LIN {X -15.567,Y 120.221,Z 250.000,A 0.000,B 0.000,C 180.000,E1 0.000} C_DIS
LIN {X -9.353,Y 120.863,Z 250.000,A 0.000,B 0.000,C 180.000,E1 0.000} C_DIS
LIN {X -3.119,Y 121.185,Z 250.000,A 0.000,B 0.000,C 180.000,E1 0.000} C_DIS
LIN {X 3.119,Y 121.185,Z 250.000,A 0.000,B 0.000,C 180.000,E1 0.000} C_DIS
LIN {X 4.435,Y 121.117,Z 250.000,A 0.000,B 0.000,C 180.000,E1 0.000} C_DIS
LIN {X 121.110,Y 4.442,Z 250.000,A 0.000,B 0.000,C 180.000,E1 0.000} C_DIS
;rapid-leaky
$VEL.CP=0.3
LIN {X 123.797,Y -61.877,Z 260.000,A 0.000,B 0.000,C 180.000,E1 0.000} C_DIS
;bead-perimeter_outer
$VEL.CP=0.29
LIN {X 126.817,Y -55.423,Z 260.000,A 0.000,B 0.000,C 180.000,E1 0.000} C_DIS
LIN {X 129.503,Y -48.820,Z 260.000,A 0.000,B 0.000,C 180.000,E1 0.000} C_DIS
LIN {X 131.844,Y -42.089,Z 260.000,A 0.000,B 0.000,C 180.000,E1 0.000} C_DIS
LIN {X 133.836,Y -35.246,Z 260.000,A 0.000,B 0.000,C 180.000,E1 0.000} C_DIS
LIN {X 135.473,Y -28.310,Z 260.000,A 0.000,B 0.000,C 180.000,E1 0.000} C_DIS
LIN {X 136.751,Y -21.298,Z 260.000,A 0.000,B 0.000,C 180.000,E1 0.000} C_DIS
LIN {X 137.666,Y -14.230,Z 260.000,A 0.000,B 0.000,C 180.000,E1 0.000} C_DIS
LIN {X 138.216,Y -7.125,Z 260.000,A 0.000,B 0.000,C 180.000,E1 0.000} C_DIS
LIN {X 138.399,Y 0.000,Z 260.000,A 0.000,B 0.000,C 180.000,E1 0.000} C_DIS
LIN {X 138.216,Y 7.125,Z 260.000,A 0.000,B 0.000,C 180.000,E1 0.000} C_DIS
LIN {X 137.666,Y 14.230,Z 260.000,A 0.000,B 0.000,C 180.000,E1 0.000} C_DIS
LIN {X 136.751,Y 21.298,Z 260.000,A 0.000,B 0.000,C 180.000,E1 0.000} C_DIS
LIN {X 135.473,Y 28.310,Z 260.000,A 0.000,B 0.000,C 180.000,E1 0.000} C_DIS
LIN {X 133.836,Y 35.246,Z 260.000,A 0.000,B 0.000,C 180.000,E1 0.000} C_DIS
LIN {X 131.844,Y 42.089,Z 260.000,A 0.000,B 0.000,C 180.000,E1 0.000} C_DIS
LIN {X 129.503,Y 48.820,Z 260.000,A 0.000,B 0.000,C 180.000,E1 0.000} C_DIS
LIN {X 126.817,Y 55.423,Z 260.000,A 0.000,B 0.000,C 180.000,E1 0.000} C_DIS
LIN {X 123.798,Y 61.876,Z 260.000,A 0.000,B 0.000,C 180.000,E1 0.000} C_DIS
LIN {X 120.447,Y 68.168,Z 260.000,A 0.000,B 0.000,C 180.000,E1 0.000} C_DIS
LIN {X 116.778,Y 74.279,Z 260.000,A 0.000,B 0.000,C 180.000,E1 0.000} C_DIS
LIN {X 112.799,Y 80.191,Z 260.000,A 0.000,B 0.000,C 180.000,E1 0.000} C_DIS
LIN {X 108.521,Y 85.892,Z 260.000,A 0.000,B 0.000,C 180.000,E1 0.000} C_DIS
LIN {X 103.956,Y 91.365,Z 260.000,A 0.000,B 0.000,C 180.000,E1 0.000} C_DIS
LIN {X 99.115,Y 96.595,Z 260.000,A 0.000,B 0.000,C 180.000,E1 0.000} C_DIS
LIN {X 94.012,Y 101.569,Z 260.000,A 0.000,B 0.000,C 180.000,E1 0.000} C_DIS
LIN {X 88.657,Y 106.273,Z 260.000,A 0.000,B 0.000,C 180.000,E1 0.000} C_DIS
LIN {X 83.069,Y 110.697,Z 260.000,A 0.000,B 0.000,C 180.000,E1 0.000} C_DIS
LIN {X 77.260,Y 114.827,Z 260.000,A 0.000,B 0.000,C 180.000,E1 0.000} C_DIS
LIN {X 71.246,Y 118.652,Z 260.000,A 0.000,B 0.000,C 180.000,E1 0.000} C_DIS
LIN {X 65.044,Y 122.163,Z 260.000,A 0.000,B 0.000,C 180.000,E1 0.000} C_DIS
LIN {X 58.671,Y 125.348,Z 260.000,A 0.000,B 0.000,C 180.000,E1 0.000} C_DIS
LIN {X 52.139,Y 128.202,Z 260.000,A 0.000,B 0.000,C 180.000,E1 0.000} C_DIS
LIN {X 45.470,Y 130.717,Z 260.000,A 0.000,B 0.000,C 180.000,E1 0.000} C_DIS
LIN {X 38.681,Y 132.884,Z 260.000,A 0.000,B 0.000,C 180.000,E1 0.000} C_DIS
LIN {X 31.788,Y 134.699,Z 260.000,A 0.000,B 0.000,C 180.000,E1 0.000} C_DIS
LIN {X 24.813,Y 136.157,Z 260.000,A 0.000,B 0.000,C 180.000,E1 0.000} C_DIS
LIN {X 17.771,Y 137.253,Z 260.000,A 0.000,B 0.000,C 180.000,E1 0.000} C_DIS
LIN {X 10.681,Y 137.986,Z 260.000,A 0.000,B 0.000,C 180.000,E1 0.000} C_DIS
LIN {X 3.564,Y 138.353,Z 260.000,A 0.000,B 0.000,C 180.000,E1 0.000} C_DIS
LIN {X -3.565,Y 138.353,Z 260.000,A 0.000,B 0.000,C 180.000,E1 0.000} C_DIS
LIN {X -10.680,Y 137.987,Z 260.000,A 0.000,B 0.000,C 180.000,E1 0.000} C_DIS
LIN {X -17.771,Y 137.253,Z 260.000,A 0.000,B 0.000,C 180.000,E1 0.000} C_DIS
LIN {X -24.813,Y 136.157,Z 260.000,A 0.000,B 0.000,C 180.000,E1 0.000} C_DIS
LIN {X -31.788,Y 134.699,Z 260.000,A 0.000,B 0.000,C 180.000,E1 0.000} C_DIS
LIN {X -38.681,Y 132.884,Z 260.000,A 0.000,B 0.000,C 180.000,E1 0.000} C_DIS
LIN {X -45.470,Y 130.717,Z 260.000,A 0.000,B 0.000,C 180.000,E1 0.000} C_DIS
LIN {X -52.139,Y 128.202,Z 260.000,A 0.000,B 0.000,C 180.000,E1 0.000} C_DIS
LIN {X -58.671,Y 125.348,Z 260.000,A 0.000,B 0.000,C 180.000,E1 0.000} C_DIS
LIN {X -65.044,Y 122.163,Z 260.000,A 0.000,B 0.000,C 180.000,E1 0.000} C_DIS
LIN {X -71.246,Y 118.652,Z 260.000,A 0.000,B 0.000,C 180.000,E1 0.000} C_DIS
LIN {X -77.260,Y 114.827,Z 260.000,A 0.000,B 0.000,C 180.000,E1 0.000} C_DIS
LIN {X -83.069,Y 110.697,Z 260.000,A 0.000,B 0.000,C 180.000,E1 0.000} C_DIS
LIN {X -88.657,Y 106.273,Z 260.000,A 0.000,B 0.000,C 180.000,E1 0.000} C_DIS
LIN {X -94.012,Y 101.569,Z 260.000,A 0.000,B 0.000,C 180.000,E1 0.000} C_DIS
LIN {X -99.115,Y 96.595,Z 260.000,A 0.000,B 0.000,C 180.000,E1 0.000} C_DIS
LIN {X -103.956,Y 91.365,Z 260.000,A 0.000,B 0.000,C 180.000,E1 0.000} C_DIS
LIN {X -108.521,Y 85.892,Z 260.000,A 0.000,B 0.000,C 180.000,E1 0.000} C_DIS
LIN {X -112.799,Y 80.191,Z 260.000,A 0.000,B 0.000,C 180.000,E1 0.000} C_DIS
LIN {X -116.778,Y 74.278,Z 260.000,A 0.000,B 0.000,C 180.000,E1 0.000} C_DIS
LIN {X -120.446,Y 68.169,Z 260.000,A 0.000,B 0.000,C 180.000,E1 0.000} C_DIS
LIN {X -123.797,Y 61.877,Z 260.000,A 0.000,B 0.000,C 180.000,E1 0.000} C_DIS
LIN {X -126.817,Y 55.423,Z 260.000,A 0.000,B 0.000,C 180.000,E1 0.000} C_DIS
LIN {X -129.503,Y 48.820,Z 260.000,A 0.000,B 0.000,C 180.000,E1 0.000} C_DIS
LIN {X -131.844,Y 42.089,Z 260.000,A 0.000,B 0.000,C 180.000,E1 0.000} C_DIS
LIN {X -133.836,Y 35.246,Z 260.000,A 0.000,B 0.000,C 180.000,E1 0.000} C_DIS
LIN {X -135.473,Y 28.310,Z 260.000,A 0.000,B 0.000,C 180.000,E1 0.000} C_DIS
LIN {X -136.751,Y 21.298,Z 260.000,A 0.000,B 0.000,C 180.000,E1 0.000} C_DIS
LIN {X -137.666,Y 14.230,Z 260.000,A 0.000,B 0.000,C 180.000,E1 0.000} C_DIS
LIN {X -138.216,Y 7.125,Z 260.000,A 0.000,B 0.000,C 180.000,E1 0.000} C_DIS
LIN {X -138.399,Y 0.000,Z 260.000,A 0.000,B 0.000,C 180.000,E1 0.000} C_DIS
LIN {X -138.216,Y -7.125,Z 260.000,A 0.000,B 0.000,C 180.000,E1 0.000} C_DIS
LIN {X -137.666,Y -14.230,Z 260.000,A 0.000,B 0.000,C 180.000,E1 0.000} C_DIS
LIN {X -136.751,Y -21.298,Z 260.000,A 0.000,B 0.000,C 180.000,E1 0.000} C_DIS
LIN {X -135.473,Y -28.310,Z 260.000,A 0.000,B 0.000,C 180.000,E1 0.000} C_DIS
LIN {X -133.836,Y -35.246,Z 260.000,A 0.000,B 0.000,C 180.000,E1 0.000} C_DIS
LIN {X -131.844,Y -42.089,Z 260.000,A 0.000,B 0.000,C 180.000,E1 0.000} C_DIS
LIN {X -129.503,Y -48.820,Z 260.000,A 0.000,B 0.000,C 180.000,E1 0.000} C_DIS
LIN {X -126.817,Y -55.423,Z 260.000,A 0.000,B 0.000,C 180.000,E1 0.000} C_DIS
LIN {X -123.798,Y -61.876,Z 260.000,A 0.000,B 0.000,C 180.000,E1 0.000} C_DIS
LIN {X -120.447,Y -68.168,Z 260.000,A 0.000,B 0.000,C 180.000,E1 0.000} C_DIS
LIN {X -116.778,Y -74.279,Z 260.000,A 0.000,B 0.000,C 180.000,E1 0.000} C_DIS
LIN {X -112.799,Y -80.191,Z 260.000,A 0.000,B 0.000,C 180.000,E1 0.000} C_DIS
LIN {X -108.521,Y -85.892,Z 260.000,A 0.000,B 0.000,C 180.000,E1 0.000} C_DIS
LIN {X -103.956,Y -91.365,Z 260.000,A 0.000,B 0.000,C 180.000,E1 0.000} C_DIS
LIN {X -99.115,Y -96.595,Z 260.000,A 0.000,B 0.000,C 180.000,E1 0.000} C_DIS
LIN {X -94.012,Y -101.569,Z 260.000,A 0.000,B 0.000,C 180.000,E1 0.000} C_DIS
LIN {X -88.657,Y -106.273,Z 260.000,A 0.000,B 0.000,C 180.000,E1 0.000} C_DIS
LIN {X -83.069,Y -110.697,Z 260.000,A 0.000,B 0.000,C 180.000,E1 0.000} C_DIS
LIN {X -77.260,Y -114.827,Z 260.000,A 0.000,B 0.000,C 180.000,E1 0.000} C_DIS
LIN {X -71.246,Y -118.652,Z 260.000,A 0.000,B 0.000,C 180.000,E1 0.000} C_DIS
LIN {X -65.044,Y -122.163,Z 260.000,A 0.000,B 0.000,C 180.000,E1 0.000} C_DIS
LIN {X -58.671,Y -125.348,Z 260.000,A 0.000,B 0.000,C 180.000,E1 0.000} C_DIS
LIN {X -52.139,Y -128.202,Z 260.000,A 0.000,B 0.000,C 180.000,E1 0.000} C_DIS
LIN {X -45.470,Y -130.717,Z 260.000,A 0.000,B 0.000,C 180.000,E1 0.000} C_DIS
LIN {X -38.681,Y -132.884,Z 260.000,A 0.000,B 0.000,C 180.000,E1 0.000} C_DIS
LIN {X -31.788,Y -134.699,Z 260.000,A 0.000,B 0.000,C 180.000,E1 0.000} C_DIS
LIN {X -24.813,Y -136.157,Z 260.000,A 0.000,B 0.000,C 180.000,E1 0.000} C_DIS
LIN {X -17.771,Y -137.253,Z 260.000,A 0.000,B 0.000,C 180.000,E1 0.000} C_DIS
LIN {X -10.681,Y -137.986,Z 260.000,A 0.000,B 0.000,C 180.000,E1 0.000} C_DIS
LIN {X -3.564,Y -138.353,Z 260.000,A 0.000,B 0.000,C 180.000,E1 0.000} C_DIS
LIN {X 3.565,Y -138.353,Z 260.000,A 0.000,B 0.000,C 180.000,E1 0.000} C_DIS
LIN {X 10.680,Y -137.987,Z 260.000,A 0.000,B 0.000,C 180.000,E1 0.000} C_DIS
LIN {X 17.771,Y -137.253,Z 260.000,A 0.000,B 0.000,C 180.000,E1 0.000} C_DIS
LIN {X 24.813,Y -136.157,Z 260.000,A 0.000,B 0.000,C 180.000,E1 0.000} C_DIS
LIN {X 31.788,Y -134.699,Z 260.000,A 0.000,B 0.000,C 180.000,E1 0.000} C_DIS
LIN {X 38.681,Y -132.884,Z 260.000,A 0.000,B 0.000,C 180.000,E1 0.000} C_DIS
LIN {X 45.470,Y -130.717,Z 260.000,A 0.000,B 0.000,C 180.000,E1 0.000} C_DIS
LIN {X 52.139,Y -128.202,Z 260.000,A 0.000,B 0.000,C 180.000,E1 0.000} C_DIS
LIN {X 58.671,Y -125.348,Z 260.000,A 0.000,B 0.000,C 180.000,E1 0.000} C_DIS
LIN {X 65.044,Y -122.163,Z 260.000,A 0.000,B 0.000,C 180.000,E1 0.000} C_DIS
LIN {X 71.246,Y -118.652,Z 260.000,A 0.000,B 0.000,C 180.000,E1 0.000} C_DIS
LIN {X 77.260,Y -114.827,Z 260.000,A 0.000,B 0.000,C 180.000,E1 0.000} C_DIS
LIN {X 83.069,Y -110.697,Z 260.000,A 0.000,B 0.000,C 180.000,E1 0.000} C_DIS
LIN {X 88.657,Y -106.273,Z 260.000,A 0.000,B 0.000,C 180.000,E1 0.000} C_DIS
LIN {X 94.012,Y -101.569,Z 260.000,A 0.000,B 0.000,C 180.000,E1 0.000} C_DIS
LIN {X 99.115,Y -96.595,Z 260.000,A 0.000,B 0.000,C 180.000,E1 0.000} C_DIS
LIN {X 103.956,Y -91.365,Z 260.000,A 0.000,B 0.000,C 180.000,E1 0.000} C_DIS
LIN {X 108.521,Y -85.892,Z 260.000,A 0.000,B 0.000,C 180.000,E1 0.000} C_DIS
LIN {X 112.799,Y -80.191,Z 260.000,A 0.000,B 0.000,C 180.000,E1 0.000} C_DIS
LIN {X 116.778,Y -74.278,Z 260.000,A 0.000,B 0.000,C 180.000,E1 0.000} C_DIS
LIN {X 120.446,Y -68.169,Z 260.000,A 0.000,B 0.000,C 180.000,E1 0.000} C_DIS
LIN {X 123.797,Y -61.877,Z 260.000,A 0.000,B 0.000,C 180.000,E1 0.000} C_DIS
;rapid-leaky
$VEL.CP=0.3
LIN {X 109.892,Y -54.927,Z 260.000,A 0.000,B 0.000,C 180.000,E1 0.000} C_DIS
;bead-perimeter_inner
$VEL.CP=0.29
LIN {X 112.573,Y -49.198,Z 260.000,A 0.000,B 0.000,C 180.000,E1 0.000} C_DIS
LIN {X 114.957,Y -43.336,Z 260.000,A 0.000,B 0.000,C 180.000,E1 0.000} C_DIS
LIN {X 117.035,Y -37.362,Z 260.000,A 0.000,B 0.000,C 180.000,E1 0.000} C_DIS
LIN {X 118.804,Y -31.287,Z 260.000,A 0.000,B 0.000,C 180.000,E1 0.000} C_DIS
LIN {X 120.256,Y -25.131,Z 260.000,A 0.000,B 0.000,C 180.000,E1 0.000} C_DIS
LIN {X 121.391,Y -18.906,Z 260.000,A 0.000,B 0.000,C 180.000,E1 0.000} C_DIS
LIN {X 122.203,Y -12.631,Z 260.000,A 0.000,B 0.000,C 180.000,E1 0.000} C_DIS
LIN {X 122.691,Y -6.325,Z 260.000,A 0.000,B 0.000,C 180.000,E1 0.000} C_DIS
LIN {X 122.854,Y 0.000,Z 260.000,A 0.000,B 0.000,C 180.000,E1 0.000} C_DIS
LIN {X 122.691,Y 6.325,Z 260.000,A 0.000,B 0.000,C 180.000,E1 0.000} C_DIS
LIN {X 122.203,Y 12.631,Z 260.000,A 0.000,B 0.000,C 180.000,E1 0.000} C_DIS
LIN {X 121.391,Y 18.906,Z 260.000,A 0.000,B 0.000,C 180.000,E1 0.000} C_DIS
LIN {X 120.256,Y 25.131,Z 260.000,A 0.000,B 0.000,C 180.000,E1 0.000} C_DIS
LIN {X 118.804,Y 31.287,Z 260.000,A 0.000,B 0.000,C 180.000,E1 0.000} C_DIS
LIN {X 117.035,Y 37.362,Z 260.000,A 0.000,B 0.000,C 180.000,E1 0.000} C_DIS
LIN {X 114.957,Y 43.336,Z 260.000,A 0.000,B 0.000,C 180.000,E1 0.000} C_DIS
LIN {X 112.572,Y 49.199,Z 260.000,A 0.000,B 0.000,C 180.000,E1 0.000} C_DIS
LIN {X 109.894,Y 54.923,Z 260.000,A 0.000,B 0.000,C 180.000,E1 0.000} C_DIS
LIN {X 106.918,Y 60.511,Z 260.000,A 0.000,B 0.000,C 180.000,E1 0.000} C_DIS
LIN {X 103.661,Y 65.936,Z 260.000,A 0.000,B 0.000,C 180.000,E1 0.000} C_DIS
LIN {X 100.130,Y 71.184,Z 260.000,A 0.000,B 0.000,C 180.000,E1 0.000} C_DIS
LIN {X 96.331,Y 76.246,Z 260.000,A 0.000,B 0.000,C 180.000,E1 0.000} C_DIS
LIN {X 92.280,Y 81.103,Z 260.000,A 0.000,B 0.000,C 180.000,E1 0.000} C_DIS
LIN {X 87.983,Y 85.745,Z 260.000,A 0.000,B 0.000,C 180.000,E1 0.000} C_DIS
LIN {X 83.453,Y 90.160,Z 260.000,A 0.000,B 0.000,C 180.000,E1 0.000} C_DIS
LIN {X 78.700,Y 94.336,Z 260.000,A 0.000,B 0.000,C 180.000,E1 0.000} C_DIS
LIN {X 73.738,Y 98.264,Z 260.000,A 0.000,B 0.000,C 180.000,E1 0.000} C_DIS
LIN {X 68.582,Y 101.929,Z 260.000,A 0.000,B 0.000,C 180.000,E1 0.000} C_DIS
LIN {X 63.243,Y 105.326,Z 260.000,A 0.000,B 0.000,C 180.000,E1 0.000} C_DIS
LIN {X 57.738,Y 108.442,Z 260.000,A 0.000,B 0.000,C 180.000,E1 0.000} C_DIS
LIN {X 52.082,Y 111.268,Z 260.000,A 0.000,B 0.000,C 180.000,E1 0.000} C_DIS
LIN {X 46.283,Y 113.803,Z 260.000,A 0.000,B 0.000,C 180.000,E1 0.000} C_DIS
LIN {X 40.363,Y 116.034,Z 260.000,A 0.000,B 0.000,C 180.000,E1 0.000} C_DIS
LIN {X 34.336,Y 117.958,Z 260.000,A 0.000,B 0.000,C 180.000,E1 0.000} C_DIS
LIN {X 28.217,Y 119.570,Z 260.000,A 0.000,B 0.000,C 180.000,E1 0.000} C_DIS
LIN {X 22.026,Y 120.864,Z 260.000,A 0.000,B 0.000,C 180.000,E1 0.000} C_DIS
LIN {X 15.775,Y 121.837,Z 260.000,A 0.000,B 0.000,C 180.000,E1 0.000} C_DIS
LIN {X 9.481,Y 122.488,Z 260.000,A 0.000,B 0.000,C 180.000,E1 0.000} C_DIS
LIN {X 3.164,Y 122.813,Z 260.000,A 0.000,B 0.000,C 180.000,E1 0.000} C_DIS
LIN {X -3.165,Y 122.813,Z 260.000,A 0.000,B 0.000,C 180.000,E1 0.000} C_DIS
LIN {X -9.479,Y 122.488,Z 260.000,A 0.000,B 0.000,C 180.000,E1 0.000} C_DIS
LIN {X -15.775,Y 121.837,Z 260.000,A 0.000,B 0.000,C 180.000,E1 0.000} C_DIS
LIN {X -22.026,Y 120.864,Z 260.000,A 0.000,B 0.000,C 180.000,E1 0.000} C_DIS
LIN {X -28.217,Y 119.570,Z 260.000,A 0.000,B 0.000,C 180.000,E1 0.000} C_DIS
LIN {X -34.336,Y 117.958,Z 260.000,A 0.000,B 0.000,C 180.000,E1 0.000} C_DIS
LIN {X -40.363,Y 116.034,Z 260.000,A 0.000,B 0.000,C 180.000,E1 0.000} C_DIS
LIN {X -46.283,Y 113.803,Z 260.000,A 0.000,B 0.000,C 180.000,E1 0.000} C_DIS
LIN {X -52.082,Y 111.268,Z 260.000,A 0.000,B 0.000,C 180.000,E1 0.000} C_DIS
LIN {X -57.738,Y 108.442,Z 260.000,A 0.000,B 0.000,C 180.000,E1 0.000} C_DIS
LIN {X -63.243,Y 105.326,Z 260.000,A 0.000,B 0.000,C 180.000,E1 0.000} C_DIS
LIN {X -68.582,Y 101.929,Z 260.000,A 0.000,B 0.000,C 180.000,E1 0.000} C_DIS
LIN {X -73.738,Y 98.264,Z 260.000,A 0.000,B 0.000,C 180.000,E1 0.000} C_DIS
LIN {X -78.700,Y 94.336,Z 260.000,A 0.000,B 0.000,C 180.000,E1 0.000} C_DIS
LIN {X -83.453,Y 90.160,Z 260.000,A 0.000,B 0.000,C 180.000,E1 0.000} C_DIS
LIN {X -87.983,Y 85.745,Z 260.000,A 0.000,B 0.000,C 180.000,E1 0.000} C_DIS
LIN {X -92.280,Y 81.103,Z 260.000,A 0.000,B 0.000,C 180.000,E1 0.000} C_DIS
LIN {X -96.331,Y 76.246,Z 260.000,A 0.000,B 0.000,C 180.000,E1 0.000} C_DIS
LIN {X -100.130,Y 71.184,Z 260.000,A 0.000,B 0.000,C 180.000,E1 0.000} C_DIS
LIN {X -103.662,Y 65.935,Z 260.000,A 0.000,B 0.000,C 180.000,E1 0.000} C_DIS
LIN {X -106.917,Y 60.513,Z 260.000,A 0.000,B 0.000,C 180.000,E1 0.000} C_DIS
LIN {X -109.892,Y 54.927,Z 260.000,A 0.000,B 0.000,C 180.000,E1 0.000} C_DIS
LIN {X -112.573,Y 49.198,Z 260.000,A 0.000,B 0.000,C 180.000,E1 0.000} C_DIS
LIN {X -114.957,Y 43.336,Z 260.000,A 0.000,B 0.000,C 180.000,E1 0.000} C_DIS
LIN {X -117.035,Y 37.362,Z 260.000,A 0.000,B 0.000,C 180.000,E1 0.000} C_DIS
LIN {X -118.804,Y 31.287,Z 260.000,A 0.000,B 0.000,C 180.000,E1 0.000} C_DIS
LIN {X -120.256,Y 25.131,Z 260.000,A 0.000,B 0.000,C 180.000,E1 0.000} C_DIS
LIN {X -121.391,Y 18.906,Z 260.000,A 0.000,B 0.000,C 180.000,E1 0.000} C_DIS
LIN {X -122.203,Y 12.631,Z 260.000,A 0.000,B 0.000,C 180.000,E1 0.000} C_DIS
LIN {X -122.691,Y 6.325,Z 260.000,A 0.000,B 0.000,C 180.000,E1 0.000} C_DIS
LIN {X -122.854,Y 0.000,Z 260.000,A 0.000,B 0.000,C 180.000,E1 0.000} C_DIS
LIN {X -122.691,Y -6.325,Z 260.000,A 0.000,B 0.000,C 180.000,E1 0.000} C_DIS
LIN {X -122.203,Y -12.631,Z 260.000,A 0.000,B 0.000,C 180.000,E1 0.000} C_DIS
LIN {X -121.391,Y -18.906,Z 260.000,A 0.000,B 0.000,C 180.000,E1 0.000} C_DIS
LIN {X -120.256,Y -25.131,Z 260.000,A 0.000,B 0.000,C 180.000,E1 0.000} C_DIS
LIN {X -118.804,Y -31.287,Z 260.000,A 0.000,B 0.000,C 180.000,E1 0.000} C_DIS
LIN {X -117.035,Y -37.362,Z 260.000,A 0.000,B 0.000,C 180.000,E1 0.000} C_DIS
LIN {X -114.957,Y -43.336,Z 260.000,A 0.000,B 0.000,C 180.000,E1 0.000} C_DIS
LIN {X -112.572,Y -49.199,Z 260.000,A 0.000,B 0.000,C 180.000,E1 0.000} C_DIS
LIN {X -109.894,Y -54.923,Z 260.000,A 0.000,B 0.000,C 180.000,E1 0.000} C_DIS
LIN {X -106.918,Y -60.511,Z 260.000,A 0.000,B 0.000,C 180.000,E1 0.000} C_DIS
LIN {X -103.661,Y -65.936,Z 260.000,A 0.000,B 0.000,C 180.000,E1 0.000} C_DIS
LIN {X -100.130,Y -71.184,Z 260.000,A 0.000,B 0.000,C 180.000,E1 0.000} C_DIS
LIN {X -96.331,Y -76.246,Z 260.000,A 0.000,B 0.000,C 180.000,E1 0.000} C_DIS
LIN {X -92.280,Y -81.103,Z 260.000,A 0.000,B 0.000,C 180.000,E1 0.000} C_DIS
LIN {X -87.983,Y -85.745,Z 260.000,A 0.000,B 0.000,C 180.000,E1 0.000} C_DIS
LIN {X -83.453,Y -90.160,Z 260.000,A 0.000,B 0.000,C 180.000,E1 0.000} C_DIS
LIN {X -78.700,Y -94.336,Z 260.000,A 0.000,B 0.000,C 180.000,E1 0.000} C_DIS
LIN {X -73.738,Y -98.264,Z 260.000,A 0.000,B 0.000,C 180.000,E1 0.000} C_DIS
LIN {X -68.582,Y -101.929,Z 260.000,A 0.000,B 0.000,C 180.000,E1 0.000} C_DIS
LIN {X -63.243,Y -105.326,Z 260.000,A 0.000,B 0.000,C 180.000,E1 0.000} C_DIS
LIN {X -57.738,Y -108.442,Z 260.000,A 0.000,B 0.000,C 180.000,E1 0.000} C_DIS
LIN {X -52.082,Y -111.268,Z 260.000,A 0.000,B 0.000,C 180.000,E1 0.000} C_DIS
LIN {X -46.283,Y -113.803,Z 260.000,A 0.000,B 0.000,C 180.000,E1 0.000} C_DIS
LIN {X -40.363,Y -116.034,Z 260.000,A 0.000,B 0.000,C 180.000,E1 0.000} C_DIS
LIN {X -34.336,Y -117.958,Z 260.000,A 0.000,B 0.000,C 180.000,E1 0.000} C_DIS
LIN {X -28.217,Y -119.570,Z 260.000,A 0.000,B 0.000,C 180.000,E1 0.000} C_DIS
LIN {X -22.026,Y -120.864,Z 260.000,A 0.000,B 0.000,C 180.000,E1 0.000} C_DIS
LIN {X -15.775,Y -121.837,Z 260.000,A 0.000,B 0.000,C 180.000,E1 0.000} C_DIS
LIN {X -9.481,Y -122.488,Z 260.000,A 0.000,B 0.000,C 180.000,E1 0.000} C_DIS
LIN {X -3.164,Y -122.813,Z 260.000,A 0.000,B 0.000,C 180.000,E1 0.000} C_DIS
LIN {X 3.165,Y -122.813,Z 260.000,A 0.000,B 0.000,C 180.000,E1 0.000} C_DIS
LIN {X 9.479,Y -122.488,Z 260.000,A 0.000,B 0.000,C 180.000,E1 0.000} C_DIS
LIN {X 15.775,Y -121.837,Z 260.000,A 0.000,B 0.000,C 180.000,E1 0.000} C_DIS
LIN {X 22.026,Y -120.864,Z 260.000,A 0.000,B 0.000,C 180.000,E1 0.000} C_DIS
LIN {X 28.217,Y -119.570,Z 260.000,A 0.000,B 0.000,C 180.000,E1 0.000} C_DIS
LIN {X 34.336,Y -117.958,Z 260.000,A 0.000,B 0.000,C 180.000,E1 0.000} C_DIS
LIN {X 40.363,Y -116.034,Z 260.000,A 0.000,B 0.000,C 180.000,E1 0.000} C_DIS
LIN {X 46.283,Y -113.803,Z 260.000,A 0.000,B 0.000,C 180.000,E1 0.000} C_DIS
LIN {X 52.082,Y -111.268,Z 260.000,A 0.000,B 0.000,C 180.000,E1 0.000} C_DIS
LIN {X 57.738,Y -108.442,Z 260.000,A 0.000,B 0.000,C 180.000,E1 0.000} C_DIS
LIN {X 63.243,Y -105.326,Z 260.000,A 0.000,B 0.000,C 180.000,E1 0.000} C_DIS
LIN {X 68.582,Y -101.929,Z 260.000,A 0.000,B 0.000,C 180.000,E1 0.000} C_DIS
LIN {X 73.738,Y -98.264,Z 260.000,A 0.000,B 0.000,C 180.000,E1 0.000} C_DIS
LIN {X 78.700,Y -94.336,Z 260.000,A 0.000,B 0.000,C 180.000,E1 0.000} C_DIS
LIN {X 83.453,Y -90.160,Z 260.000,A 0.000,B 0.000,C 180.000,E1 0.000} C_DIS
LIN {X 87.983,Y -85.745,Z 260.000,A 0.000,B 0.000,C 180.000,E1 0.000} C_DIS
LIN {X 92.280,Y -81.103,Z 260.000,A 0.000,B 0.000,C 180.000,E1 0.000} C_DIS
LIN {X 96.331,Y -76.246,Z 260.000,A 0.000,B 0.000,C 180.000,E1 0.000} C_DIS
LIN {X 100.130,Y -71.184,Z 260.000,A 0.000,B 0.000,C 180.000,E1 0.000} C_DIS
LIN {X 103.662,Y -65.935,Z 260.000,A 0.000,B 0.000,C 180.000,E1 0.000} C_DIS
LIN {X 106.917,Y -60.513,Z 260.000,A 0.000,B 0.000,C 180.000,E1 0.000} C_DIS
LIN {X 109.892,Y -54.927,Z 260.000,A 0.000,B 0.000,C 180.000,E1 0.000} C_DIS
;rapid-leaky
$VEL.CP=0.3
LIN {X 102.499,Y -23.053,Z 260.000,A 0.000,B 0.000,C 180.000,E1 0.000} C_DIS
;bead-sparse_infill
$VEL.CP=0.29
LIN {X 23.045,Y -102.507,Z 260.000,A 0.000,B 0.000,C 180.000,E1 0.000} C_DIS
LIN {X 18.842,Y -103.386,Z 260.000,A 0.000,B 0.000,C 180.000,E1 0.000} C_DIS
LIN {X 13.494,Y -104.218,Z 260.000,A 0.000,B 0.000,C 180.000,E1 0.000} C_DIS
LIN {X 8.108,Y -104.775,Z 260.000,A 0.000,B 0.000,C 180.000,E1 0.000} C_DIS
LIN {X 2.708,Y -105.053,Z 260.000,A 0.000,B 0.000,C 180.000,E1 0.000} C_DIS
LIN {X -2.707,Y -105.053,Z 260.000,A 0.000,B 0.000,C 180.000,E1 0.000} C_DIS
LIN {X -8.110,Y -104.775,Z 260.000,A 0.000,B 0.000,C 180.000,E1 0.000} C_DIS
LIN {X -13.494,Y -104.218,Z 260.000,A 0.000,B 0.000,C 180.000,E1 0.000} C_DIS
LIN {X -18.842,Y -103.386,Z 260.000,A 0.000,B 0.000,C 180.000,E1 0.000} C_DIS
LIN {X -24.136,Y -102.279,Z 260.000,A 0.000,B 0.000,C 180.000,E1 0.000} C_DIS
LIN {X -29.371,Y -100.900,Z 260.000,A 0.000,B 0.000,C 180.000,E1 0.000} C_DIS
LIN {X -34.526,Y -99.255,Z 260.000,A 0.000,B 0.000,C 180.000,E1 0.000} C_DIS
LIN {X -39.590,Y -97.346,Z 260.000,A 0.000,B 0.000,C 180.000,E1 0.000} C_DIS
LIN {X -44.551,Y -95.177,Z 260.000,A 0.000,B 0.000,C 180.000,E1 0.000} C_DIS
LIN {X -49.389,Y -92.760,Z 260.000,A 0.000,B 0.000,C 180.000,E1 0.000} C_DIS
LIN {X -54.096,Y -90.095,Z 260.000,A 0.000,B 0.000,C 180.000,E1 0.000} C_DIS
LIN {X -58.665,Y -87.189,Z 260.000,A 0.000,B 0.000,C 180.000,E1 0.000} C_DIS
LIN {X -63.074,Y -84.054,Z 260.000,A 0.000,B 0.000,C 180.000,E1 0.000} C_DIS
LIN {X -67.320,Y -80.694,Z 260.000,A 0.000,B 0.000,C 180.000,E1 0.000} C_DIS
LIN {X -71.386,Y -77.121,Z 260.000,A 0.000,B 0.000,C 180.000,E1 0.000} C_DIS
LIN {X -75.260,Y -73.346,Z 260.000,A 0.000,B 0.000,C 180.000,E1 0.000} C_DIS
LIN {X -78.935,Y -69.375,Z 260.000,A 0.000,B 0.000,C 180.000,E1 0.000} C_DIS
LIN {X -82.400,Y -65.221,Z 260.000,A 0.000,B 0.000,C 180.000,E1 0.000} C_DIS
LIN {X -85.650,Y -60.889,Z 260.000,A 0.000,B 0.000,C 180.000,E1 0.000} C_DIS
LIN {X -88.331,Y -56.905,Z 260.000,A 0.000,B 0.000,C 180.000,E1 0.000} C_DIS
LIN {X 56.891,Y 88.317,Z 260.000,A 0.000,B 0.000,C 180.000,E1 0.000} C_DIS
;rapid-leaky
$VEL.CP=0.3
LIN {X 93.706,Y -74.165,Z 270.000,A 0.000,B 0.000,C 180.000,E1 0.000} C_DIS
;bead-perimeter_outer
$VEL.CP=0.21
LIN {X 97.399,Y -69.244,Z 270.000,A 0.000,B 0.000,C 180.000,E1 0.000} C_DIS
LIN {X 100.834,Y -64.137,Z 270.000,A 0.000,B 0.000,C 180.000,E1 0.000} C_DIS
LIN {X 104.003,Y -58.861,Z 270.000,A 0.000,B 0.000,C 180.000,E1 0.000} C_DIS
LIN {X 106.895,Y -53.430,Z 270.000,A 0.000,B 0.000,C 180.000,E1 0.000} C_DIS
LIN {X 109.504,Y -47.856,Z 270.000,A 0.000,B 0.000,C 180.000,E1 0.000} C_DIS
LIN {X 111.822,Y -42.155,Z 270.000,A 0.000,B 0.000,C 180.000,E1 0.000} C_DIS
LIN {X 113.844,Y -36.344,Z 270.000,A 0.000,B 0.000,C 180.000,E1 0.000} C_DIS
LIN {X 115.563,Y -30.435,Z 270.000,A 0.000,B 0.000,C 180.000,E1 0.000} C_DIS
LIN {X 116.977,Y -24.445,Z 270.000,A 0.000,B 0.000,C 180.000,E1 0.000} C_DIS
LIN {X 118.080,Y -18.390,Z 270.000,A 0.000,B 0.000,C 180.000,E1 0.000} C_DIS
LIN {X 118.870,Y -12.288,Z 270.000,A 0.000,B 0.000,C 180.000,E1 0.000} C_DIS
LIN {X 119.346,Y -6.144,Z 270.000,A 0.000,B 0.000,C 180.000,E1 0.000} C_DIS
LIN {X 119.356,Y -5.765,Z 270.000,A 0.000,B 0.000,C 180.000,E1 0.000} C_DIS
LIN {X 119.503,Y -0.001,Z 270.000,A 0.000,B 0.000,C 180.000,E1 0.000} C_DIS
LIN {X 119.345,Y 6.152,Z 270.000,A 0.000,B 0.000,C 180.000,E1 0.000} C_DIS
LIN {X 118.870,Y 12.288,Z 270.000,A 0.000,B 0.000,C 180.000,E1 0.000} C_DIS
LIN {X 118.080,Y 18.390,Z 270.000,A 0.000,B 0.000,C 180.000,E1 0.000} C_DIS
LIN {X 116.977,Y 24.445,Z 270.000,A 0.000,B 0.000,C 180.000,E1 0.000} C_DIS
LIN {X 115.563,Y 30.435,Z 270.000,A 0.000,B 0.000,C 180.000,E1 0.000} C_DIS
LIN {X 113.844,Y 36.344,Z 270.000,A 0.000,B 0.000,C 180.000,E1 0.000} C_DIS
LIN {X 111.822,Y 42.155,Z 270.000,A 0.000,B 0.000,C 180.000,E1 0.000} C_DIS
LIN {X 109.504,Y 47.856,Z 270.000,A 0.000,B 0.000,C 180.000,E1 0.000} C_DIS
LIN {X 106.895,Y 53.430,Z 270.000,A 0.000,B 0.000,C 180.000,E1 0.000} C_DIS
LIN {X 104.003,Y 58.861,Z 270.000,A 0.000,B 0.000,C 180.000,E1 0.000} C_DIS
LIN {X 100.834,Y 64.137,Z 270.000,A 0.000,B 0.000,C 180.000,E1 0.000} C_DIS
LIN {X 97.399,Y 69.244,Z 270.000,A 0.000,B 0.000,C 180.000,E1 0.000} C_DIS
LIN {X 93.706,Y 74.165,Z 270.000,A 0.000,B 0.000,C 180.000,E1 0.000} C_DIS
LIN {X 89.762,Y 78.891,Z 270.000,A 0.000,B 0.000,C 180.000,E1 0.000} C_DIS
LIN {X 85.583,Y 83.407,Z 270.000,A 0.000,B 0.000,C 180.000,E1 0.000} C_DIS
LIN {X 81.176,Y 87.702,Z 270.000,A 0.000,B 0.000,C 180.000,E1 0.000} C_DIS
LIN {X 76.553,Y 91.765,Z 270.000,A 0.000,B 0.000,C 180.000,E1 0.000} C_DIS
LIN {X 71.727,Y 95.584,Z 270.000,A 0.000,B 0.000,C 180.000,E1 0.000} C_DIS
LIN {X 66.712,Y 99.150,Z 270.000,A 0.000,B 0.000,C 180.000,E1 0.000} C_DIS
LIN {X 61.520,Y 102.453,Z 270.000,A 0.000,B 0.000,C 180.000,E1 0.000} C_DIS
LIN {X 56.163,Y 105.484,Z 270.000,A 0.000,B 0.000,C 180.000,E1 0.000} C_DIS
LIN {X 50.660,Y 108.235,Z 270.000,A 0.000,B 0.000,C 180.000,E1 0.000} C_DIS
LIN {X 45.022,Y 110.699,Z 270.000,A 0.000,B 0.000,C 180.000,E1 0.000} C_DIS
LIN {X 39.262,Y 112.870,Z 270.000,A 0.000,B 0.000,C 180.000,E1 0.000} C_DIS
LIN {X 33.399,Y 114.742,Z 270.000,A 0.000,B 0.000,C 180.000,E1 0.000} C_DIS
LIN {X 27.448,Y 116.309,Z 270.000,A 0.000,B 0.000,C 180.000,E1 0.000} C_DIS
LIN {X 21.424,Y 117.568,Z 270.000,A 0.000,B 0.000,C 180.000,E1 0.000} C_DIS
LIN {X 15.345,Y 118.515,Z 270.000,A 0.000,B 0.000,C 180.000,E1 0.000} C_DIS
LIN {X 9.223,Y 119.147,Z 270.000,A 0.000,B 0.000,C 180.000,E1 0.000} C_DIS
LIN {X 3.077,Y 119.464,Z 270.000,A 0.000,B 0.000,C 180.000,E1 0.000} C_DIS
LIN {X -3.079,Y 119.464,Z 270.000,A 0.000,B 0.000,C 180.000,E1 0.000} C_DIS
LIN {X -3.458,Y 119.445,Z 270.000,A 0.000,B 0.000,C 180.000,E1 0.000} C_DIS
LIN {X -9.223,Y 119.147,Z 270.000,A 0.000,B 0.000,C 180.000,E1 0.000} C_DIS
LIN {X -15.345,Y 118.515,Z 270.000,A 0.000,B 0.000,C 180.000,E1 0.000} C_DIS
LIN {X -21.424,Y 117.568,Z 270.000,A 0.000,B 0.000,C 180.000,E1 0.000} C_DIS
LIN {X -27.448,Y 116.309,Z 270.000,A 0.000,B 0.000,C 180.000,E1 0.000} C_DIS
LIN {X -33.399,Y 114.742,Z 270.000,A 0.000,B 0.000,C 180.000,E1 0.000} C_DIS
LIN {X -39.262,Y 112.870,Z 270.000,A 0.000,B 0.000,C 180.000,E1 0.000} C_DIS
LIN {X -45.022,Y 110.699,Z 270.000,A 0.000,B 0.000,C 180.000,E1 0.000} C_DIS
LIN {X -50.660,Y 108.235,Z 270.000,A 0.000,B 0.000,C 180.000,E1 0.000} C_DIS
LIN {X -56.163,Y 105.484,Z 270.000,A 0.000,B 0.000,C 180.000,E1 0.000} C_DIS
LIN {X -61.520,Y 102.453,Z 270.000,A 0.000,B 0.000,C 180.000,E1 0.000} C_DIS
LIN {X -66.712,Y 99.150,Z 270.000,A 0.000,B 0.000,C 180.000,E1 0.000} C_DIS
LIN {X -71.727,Y 95.584,Z 270.000,A 0.000,B 0.000,C 180.000,E1 0.000} C_DIS
LIN {X -76.553,Y 91.765,Z 270.000,A 0.000,B 0.000,C 180.000,E1 0.000} C_DIS
LIN {X -81.176,Y 87.702,Z 270.000,A 0.000,B 0.000,C 180.000,E1 0.000} C_DIS
LIN {X -85.583,Y 83.407,Z 270.000,A 0.000,B 0.000,C 180.000,E1 0.000} C_DIS
LIN {X -89.762,Y 78.891,Z 270.000,A 0.000,B 0.000,C 180.000,E1 0.000} C_DIS
LIN {X -93.706,Y 74.165,Z 270.000,A 0.000,B 0.000,C 180.000,E1 0.000} C_DIS
LIN {X -97.399,Y 69.244,Z 270.000,A 0.000,B 0.000,C 180.000,E1 0.000} C_DIS
LIN {X -100.834,Y 64.137,Z 270.000,A 0.000,B 0.000,C 180.000,E1 0.000} C_DIS
LIN {X -104.003,Y 58.861,Z 270.000,A 0.000,B 0.000,C 180.000,E1 0.000} C_DIS
LIN {X -106.895,Y 53.430,Z 270.000,A 0.000,B 0.000,C 180.000,E1 0.000} C_DIS
LIN {X -109.504,Y 47.856,Z 270.000,A 0.000,B 0.000,C 180.000,E1 0.000} C_DIS
LIN {X -111.822,Y 42.155,Z 270.000,A 0.000,B 0.000,C 180.000,E1 0.000} C_DIS
LIN {X -113.844,Y 36.344,Z 270.000,A 0.000,B 0.000,C 180.000,E1 0.000} C_DIS
LIN {X -115.563,Y 30.435,Z 270.000,A 0.000,B 0.000,C 180.000,E1 0.000} C_DIS
LIN {X -116.977,Y 24.445,Z 270.000,A 0.000,B 0.000,C 180.000,E1 0.000} C_DIS
LIN {X -118.080,Y 18.390,Z 270.000,A 0.000,B 0.000,C 180.000,E1 0.000} C_DIS
LIN {X -118.870,Y 12.288,Z 270.000,A 0.000,B 0.000,C 180.000,E1 0.000} C_DIS
LIN {X -119.346,Y 6.144,Z 270.000,A 0.000,B 0.000,C 180.000,E1 0.000} C_DIS
LIN {X -119.356,Y 5.765,Z 270.000,A 0.000,B 0.000,C 180.000,E1 0.000} C_DIS
LIN {X -119.503,Y 0.001,Z 270.000,A 0.000,B 0.000,C 180.000,E1 0.000} C_DIS
LIN {X -119.345,Y -6.152,Z 270.000,A 0.000,B 0.000,C 180.000,E1 0.000} C_DIS
LIN {X -118.870,Y -12.288,Z 270.000,A 0.000,B 0.000,C 180.000,E1 0.000} C_DIS
LIN {X -118.080,Y -18.390,Z 270.000,A 0.000,B 0.000,C 180.000,E1 0.000} C_DIS
LIN {X -116.977,Y -24.445,Z 270.000,A 0.000,B 0.000,C 180.000,E1 0.000} C_DIS
LIN {X -115.563,Y -30.435,Z 270.000,A 0.000,B 0.000,C 180.000,E1 0.000} C_DIS
LIN {X -113.844,Y -36.344,Z 270.000,A 0.000,B 0.000,C 180.000,E1 0.000} C_DIS
LIN {X -111.822,Y -42.155,Z 270.000,A 0.000,B 0.000,C 180.000,E1 0.000} C_DIS
LIN {X -109.504,Y -47.856,Z 270.000,A 0.000,B 0.000,C 180.000,E1 0.000} C_DIS
LIN {X -106.895,Y -53.430,Z 270.000,A 0.000,B 0.000,C 180.000,E1 0.000} C_DIS
LIN {X -104.003,Y -58.861,Z 270.000,A 0.000,B 0.000,C 180.000,E1 0.000} C_DIS
LIN {X -100.834,Y -64.137,Z 270.000,A 0.000,B 0.000,C 180.000,E1 0.000} C_DIS
LIN {X -97.399,Y -69.244,Z 270.000,A 0.000,B 0.000,C 180.000,E1 0.000} C_DIS
LIN {X -93.706,Y -74.165,Z 270.000,A 0.000,B 0.000,C 180.000,E1 0.000} C_DIS
LIN {X -89.762,Y -78.891,Z 270.000,A 0.000,B 0.000,C 180.000,E1 0.000} C_DIS
LIN {X -85.583,Y -83.407,Z 270.000,A 0.000,B 0.000,C 180.000,E1 0.000} C_DIS
LIN {X -81.176,Y -87.702,Z 270.000,A 0.000,B 0.000,C 180.000,E1 0.000} C_DIS
LIN {X -76.553,Y -91.765,Z 270.000,A 0.000,B 0.000,C 180.000,E1 0.000} C_DIS
LIN {X -71.727,Y -95.584,Z 270.000,A 0.000,B 0.000,C 180.000,E1 0.000} C_DIS
LIN {X -66.712,Y -99.150,Z 270.000,A 0.000,B 0.000,C 180.000,E1 0.000} C_DIS
LIN {X -61.520,Y -102.453,Z 270.000,A 0.000,B 0.000,C 180.000,E1 0.000} C_DIS
LIN {X -56.163,Y -105.484,Z 270.000,A 0.000,B 0.000,C 180.000,E1 0.000} C_DIS
LIN {X -50.660,Y -108.235,Z 270.000,A 0.000,B 0.000,C 180.000,E1 0.000} C_DIS
LIN {X -45.022,Y -110.699,Z 270.000,A 0.000,B 0.000,C 180.000,E1 0.000} C_DIS
LIN {X -39.262,Y -112.870,Z 270.000,A 0.000,B 0.000,C 180.000,E1 0.000} C_DIS
LIN {X -33.399,Y -114.742,Z 270.000,A 0.000,B 0.000,C 180.000,E1 0.000} C_DIS
LIN {X -27.448,Y -116.309,Z 270.000,A 0.000,B 0.000,C 180.000,E1 0.000} C_DIS
LIN {X -21.424,Y -117.568,Z 270.000,A 0.000,B 0.000,C 180.000,E1 0.000} C_DIS
LIN {X -15.345,Y -118.515,Z 270.000,A 0.000,B 0.000,C 180.000,E1 0.000} C_DIS
LIN {X -9.223,Y -119.147,Z 270.000,A 0.000,B 0.000,C 180.000,E1 0.000} C_DIS
LIN {X -3.077,Y -119.464,Z 270.000,A 0.000,B 0.000,C 180.000,E1 0.000} C_DIS
LIN {X 3.079,Y -119.464,Z 270.000,A 0.000,B 0.000,C 180.000,E1 0.000} C_DIS
LIN {X 9.223,Y -119.147,Z 270.000,A 0.000,B 0.000,C 180.000,E1 0.000} C_DIS
LIN {X 15.345,Y -118.515,Z 270.000,A 0.000,B 0.000,C 180.000,E1 0.000} C_DIS
LIN {X 21.424,Y -117.568,Z 270.000,A 0.000,B 0.000,C 180.000,E1 0.000} C_DIS
LIN {X 27.448,Y -116.309,Z 270.000,A 0.000,B 0.000,C 180.000,E1 0.000} C_DIS
LIN {X 33.399,Y -114.742,Z 270.000,A 0.000,B 0.000,C 180.000,E1 0.000} C_DIS
LIN {X 39.262,Y -112.870,Z 270.000,A 0.000,B 0.000,C 180.000,E1 0.000} C_DIS
LIN {X 45.022,Y -110.699,Z 270.000,A 0.000,B 0.000,C 180.000,E1 0.000} C_DIS
LIN {X 50.660,Y -108.235,Z 270.000,A 0.000,B 0.000,C 180.000,E1 0.000} C_DIS
LIN {X 56.163,Y -105.484,Z 270.000,A 0.000,B 0.000,C 180.000,E1 0.000} C_DIS
LIN {X 61.520,Y -102.453,Z 270.000,A 0.000,B 0.000,C 180.000,E1 0.000} C_DIS
LIN {X 66.712,Y -99.150,Z 270.000,A 0.000,B 0.000,C 180.000,E1 0.000} C_DIS
LIN {X 71.727,Y -95.584,Z 270.000,A 0.000,B 0.000,C 180.000,E1 0.000} C_DIS
LIN {X 76.553,Y -91.765,Z 270.000,A 0.000,B 0.000,C 180.000,E1 0.000} C_DIS
LIN {X 81.176,Y -87.702,Z 270.000,A 0.000,B 0.000,C 180.000,E1 0.000} C_DIS
LIN {X 85.583,Y -83.407,Z 270.000,A 0.000,B 0.000,C 180.000,E1 0.000} C_DIS
LIN {X 89.762,Y -78.891,Z 270.000,A 0.000,B 0.000,C 180.000,E1 0.000} C_DIS
LIN {X 93.706,Y -74.165,Z 270.000,A 0.000,B 0.000,C 180.000,E1 0.000} C_DIS
;rapid-leaky
$VEL.CP=0.3
LIN {X 81.517,Y -64.517,Z 270.000,A 0.000,B 0.000,C 180.000,E1 0.000} C_DIS
;bead-perimeter_inner
$VEL.CP=0.21
LIN {X 84.729,Y -60.237,Z 270.000,A 0.000,B 0.000,C 180.000,E1 0.000} C_DIS
LIN {X 87.718,Y -55.794,Z 270.000,A 0.000,B 0.000,C 180.000,E1 0.000} C_DIS
LIN {X 90.475,Y -51.203,Z 270.000,A 0.000,B 0.000,C 180.000,E1 0.000} C_DIS
LIN {X 92.990,Y -46.480,Z 270.000,A 0.000,B 0.000,C 180.000,E1 0.000} C_DIS
LIN {X 95.259,Y -41.630,Z 270.000,A 0.000,B 0.000,C 180.000,E1 0.000} C_DIS
LIN {X 97.277,Y -36.670,Z 270.000,A 0.000,B 0.000,C 180.000,E1 0.000} C_DIS
LIN {X 99.035,Y -31.616,Z 270.000,A 0.000,B 0.000,C 180.000,E1 0.000} C_DIS
LIN {X 100.531,Y -26.477,Z 270.000,A 0.000,B 0.000,C 180.000,E1 0.000} C_DIS
LIN {X 101.760,Y -21.266,Z 270.000,A 0.000,B 0.000,C 180.000,E1 0.000} C_DIS
LIN {X 102.720,Y -15.999,Z 270.000,A 0.000,B 0.000,C 180.000,E1 0.000} C_DIS
LIN {X 103.407,Y -10.689,Z 270.000,A 0.000,B 0.000,C 180.000,E1 0.000} C_DIS
LIN {X 103.822,Y -5.335,Z 270.000,A 0.000,B 0.000,C 180.000,E1 0.000} C_DIS
LIN {X 103.958,Y -0.002,Z 270.000,A 0.000,B 0.000,C 180.000,E1 0.000} C_DIS
LIN {X 103.820,Y 5.352,Z 270.000,A 0.000,B 0.000,C 180.000,E1 0.000} C_DIS
LIN {X 103.407,Y 10.689,Z 270.000,A 0.000,B 0.000,C 180.000,E1 0.000} C_DIS
LIN {X 102.720,Y 15.999,Z 270.000,A 0.000,B 0.000,C 180.000,E1 0.000} C_DIS
LIN {X 101.760,Y 21.266,Z 270.000,A 0.000,B 0.000,C 180.000,E1 0.000} C_DIS
LIN {X 100.531,Y 26.477,Z 270.000,A 0.000,B 0.000,C 180.000,E1 0.000} C_DIS
LIN {X 99.035,Y 31.616,Z 270.000,A 0.000,B 0.000,C 180.000,E1 0.000} C_DIS
LIN {X 97.277,Y 36.670,Z 270.000,A 0.000,B 0.000,C 180.000,E1 0.000} C_DIS
LIN {X 95.259,Y 41.630,Z 270.000,A 0.000,B 0.000,C 180.000,E1 0.000} C_DIS
LIN {X 92.990,Y 46.480,Z 270.000,A 0.000,B 0.000,C 180.000,E1 0.000} C_DIS
LIN {X 90.475,Y 51.203,Z 270.000,A 0.000,B 0.000,C 180.000,E1 0.000} C_DIS
LIN {X 87.718,Y 55.794,Z 270.000,A 0.000,B 0.000,C 180.000,E1 0.000} C_DIS
LIN {X 84.729,Y 60.237,Z 270.000,A 0.000,B 0.000,C 180.000,E1 0.000} C_DIS
LIN {X 81.517,Y 64.517,Z 270.000,A 0.000,B 0.000,C 180.000,E1 0.000} C_DIS
LIN {X 78.086,Y 68.629,Z 270.000,A 0.000,B 0.000,C 180.000,E1 0.000} C_DIS
LIN {X 74.450,Y 72.558,Z 270.000,A 0.000,B 0.000,C 180.000,E1 0.000} C_DIS
LIN {X 70.617,Y 76.293,Z 270.000,A 0.000,B 0.000,C 180.000,E1 0.000} C_DIS
LIN {X 66.595,Y 79.828,Z 270.000,A 0.000,B 0.000,C 180.000,E1 0.000} C_DIS
LIN {X 62.397,Y 83.150,Z 270.000,A 0.000,B 0.000,C 180.000,E1 0.000} C_DIS
LIN {X 58.033,Y 86.253,Z 270.000,A 0.000,B 0.000,C 180.000,E1 0.000} C_DIS
LIN {X 53.517,Y 89.126,Z 270.000,A 0.000,B 0.000,C 180.000,E1 0.000} C_DIS
LIN {X 48.857,Y 91.763,Z 270.000,A 0.000,B 0.000,C 180.000,E1 0.000} C_DIS
LIN {X 44.070,Y 94.156,Z 270.000,A 0.000,B 0.000,C 180.000,E1 0.000} C_DIS
LIN {X 39.167,Y 96.299,Z 270.000,A 0.000,B 0.000,C 180.000,E1 0.000} C_DIS
LIN {X 34.155,Y 98.187,Z 270.000,A 0.000,B 0.000,C 180.000,E1 0.000} C_DIS
LIN {X 29.054,Y 99.817,Z 270.000,A 0.000,B 0.000,C 180.000,E1 0.000} C_DIS
LIN {X 23.878,Y 101.180,Z 270.000,A 0.000,B 0.000,C 180.000,E1 0.000} C_DIS
LIN {X 18.637,Y 102.275,Z 270.000,A 0.000,B 0.000,C 180.000,E1 0.000} C_DIS
LIN {X 13.349,Y 103.099,Z 270.000,A 0.000,B 0.000,C 180.000,E1 0.000} C_DIS
LIN {X 8.024,Y 103.649,Z 270.000,A 0.000,B 0.000,C 180.000,E1 0.000} C_DIS
LIN {X 2.677,Y 103.924,Z 270.000,A 0.000,B 0.000,C 180.000,E1 0.000} C_DIS
LIN {X -2.682,Y 103.924,Z 270.000,A 0.000,B 0.000,C 180.000,E1 0.000} C_DIS
LIN {X -8.023,Y 103.649,Z 270.000,A 0.000,B 0.000,C 180.000,E1 0.000} C_DIS
LIN {X -13.349,Y 103.099,Z 270.000,A 0.000,B 0.000,C 180.000,E1 0.000} C_DIS
LIN {X -18.637,Y 102.275,Z 270.000,A 0.000,B 0.000,C 180.000,E1 0.000} C_DIS
LIN {X -23.878,Y 101.180,Z 270.000,A 0.000,B 0.000,C 180.000,E1 0.000} C_DIS
LIN {X -29.054,Y 99.817,Z 270.000,A 0.000,B 0.000,C 180.000,E1 0.000} C_DIS
LIN {X -34.155,Y 98.187,Z 270.000,A 0.000,B 0.000,C 180.000,E1 0.000} C_DIS
LIN {X -39.167,Y 96.299,Z 270.000,A 0.000,B 0.000,C 180.000,E1 0.000} C_DIS
LIN {X -44.070,Y 94.156,Z 270.000,A 0.000,B 0.000,C 180.000,E1 0.000} C_DIS
LIN {X -48.857,Y 91.763,Z 270.000,A 0.000,B 0.000,C 180.000,E1 0.000} C_DIS
LIN {X -53.517,Y 89.126,Z 270.000,A 0.000,B 0.000,C 180.000,E1 0.000} C_DIS
LIN {X -58.033,Y 86.253,Z 270.000,A 0.000,B 0.000,C 180.000,E1 0.000} C_DIS
LIN {X -62.397,Y 83.150,Z 270.000,A 0.000,B 0.000,C 180.000,E1 0.000} C_DIS
LIN {X -66.595,Y 79.828,Z 270.000,A 0.000,B 0.000,C 180.000,E1 0.000} C_DIS
LIN {X -70.617,Y 76.293,Z 270.000,A 0.000,B 0.000,C 180.000,E1 0.000} C_DIS
LIN {X -74.450,Y 72.558,Z 270.000,A 0.000,B 0.000,C 180.000,E1 0.000} C_DIS
LIN {X -78.086,Y 68.629,Z 270.000,A 0.000,B 0.000,C 180.000,E1 0.000} C_DIS
LIN {X -81.517,Y 64.517,Z 270.000,A 0.000,B 0.000,C 180.000,E1 0.000} C_DIS
LIN {X -84.729,Y 60.237,Z 270.000,A 0.000,B 0.000,C 180.000,E1 0.000} C_DIS
LIN {X -87.718,Y 55.794,Z 270.000,A 0.000,B 0.000,C 180.000,E1 0.000} C_DIS
LIN {X -90.475,Y 51.203,Z 270.000,A 0.000,B 0.000,C 180.000,E1 0.000} C_DIS
LIN {X -92.990,Y 46.480,Z 270.000,A 0.000,B 0.000,C 180.000,E1 0.000} C_DIS
LIN {X -95.259,Y 41.630,Z 270.000,A 0.000,B 0.000,C 180.000,E1 0.000} C_DIS
LIN {X -97.277,Y 36.670,Z 270.000,A 0.000,B 0.000,C 180.000,E1 0.000} C_DIS
LIN {X -99.035,Y 31.616,Z 270.000,A 0.000,B 0.000,C 180.000,E1 0.000} C_DIS
LIN {X -100.531,Y 26.477,Z 270.000,A 0.000,B 0.000,C 180.000,E1 0.000} C_DIS
LIN {X -101.760,Y 21.266,Z 270.000,A 0.000,B 0.000,C 180.000,E1 0.000} C_DIS
LIN {X -102.720,Y 15.999,Z 270.000,A 0.000,B 0.000,C 180.000,E1 0.000} C_DIS
LIN {X -103.407,Y 10.689,Z 270.000,A 0.000,B 0.000,C 180.000,E1 0.000} C_DIS
LIN {X -103.822,Y 5.335,Z 270.000,A 0.000,B 0.000,C 180.000,E1 0.000} C_DIS
LIN {X -103.958,Y 0.002,Z 270.000,A 0.000,B 0.000,C 180.000,E1 0.000} C_DIS
LIN {X -103.820,Y -5.352,Z 270.000,A 0.000,B 0.000,C 180.000,E1 0.000} C_DIS
LIN {X -103.407,Y -10.689,Z 270.000,A 0.000,B 0.000,C 180.000,E1 0.000} C_DIS
LIN {X -102.720,Y -15.999,Z 270.000,A 0.000,B 0.000,C 180.000,E1 0.000} C_DIS
LIN {X -101.760,Y -21.266,Z 270.000,A 0.000,B 0.000,C 180.000,E1 0.000} C_DIS
LIN {X -100.531,Y -26.477,Z 270.000,A 0.000,B 0.000,C 180.000,E1 0.000} C_DIS
LIN {X -99.035,Y -31.616,Z 270.000,A 0.000,B 0.000,C 180.000,E1 0.000} C_DIS
LIN {X -97.277,Y -36.670,Z 270.000,A 0.000,B 0.000,C 180.000,E1 0.000} C_DIS
LIN {X -95.259,Y -41.630,Z 270.000,A 0.000,B 0.000,C 180.000,E1 0.000} C_DIS
LIN {X -92.990,Y -46.480,Z 270.000,A 0.000,B 0.000,C 180.000,E1 0.000} C_DIS
LIN {X -90.475,Y -51.203,Z 270.000,A 0.000,B 0.000,C 180.000,E1 0.000} C_DIS
LIN {X -87.718,Y -55.794,Z 270.000,A 0.000,B 0.000,C 180.000,E1 0.000} C_DIS
LIN {X -84.729,Y -60.237,Z 270.000,A 0.000,B 0.000,C 180.000,E1 0.000} C_DIS
LIN {X -81.517,Y -64.517,Z 270.000,A 0.000,B 0.000,C 180.000,E1 0.000} C_DIS
LIN {X -78.086,Y -68.629,Z 270.000,A 0.000,B 0.000,C 180.000,E1 0.000} C_DIS
LIN {X -74.450,Y -72.558,Z 270.000,A 0.000,B 0.000,C 180.000,E1 0.000} C_DIS
LIN {X -70.617,Y -76.293,Z 270.000,A 0.000,B 0.000,C 180.000,E1 0.000} C_DIS
LIN {X -66.595,Y -79.828,Z 270.000,A 0.000,B 0.000,C 180.000,E1 0.000} C_DIS
LIN {X -62.397,Y -83.150,Z 270.000,A 0.000,B 0.000,C 180.000,E1 0.000} C_DIS
LIN {X -58.033,Y -86.253,Z 270.000,A 0.000,B 0.000,C 180.000,E1 0.000} C_DIS
LIN {X -53.517,Y -89.126,Z 270.000,A 0.000,B 0.000,C 180.000,E1 0.000} C_DIS
LIN {X -48.857,Y -91.763,Z 270.000,A 0.000,B 0.000,C 180.000,E1 0.000} C_DIS
LIN {X -44.070,Y -94.156,Z 270.000,A 0.000,B 0.000,C 180.000,E1 0.000} C_DIS
LIN {X -39.167,Y -96.299,Z 270.000,A 0.000,B 0.000,C 180.000,E1 0.000} C_DIS
LIN {X -34.155,Y -98.187,Z 270.000,A 0.000,B 0.000,C 180.000,E1 0.000} C_DIS
LIN {X -29.054,Y -99.817,Z 270.000,A 0.000,B 0.000,C 180.000,E1 0.000} C_DIS
LIN {X -23.878,Y -101.180,Z 270.000,A 0.000,B 0.000,C 180.000,E1 0.000} C_DIS
LIN {X -18.637,Y -102.275,Z 270.000,A 0.000,B 0.000,C 180.000,E1 0.000} C_DIS
LIN {X -13.349,Y -103.099,Z 270.000,A 0.000,B 0.000,C 180.000,E1 0.000} C_DIS
LIN {X -8.024,Y -103.649,Z 270.000,A 0.000,B 0.000,C 180.000,E1 0.000} C_DIS
LIN {X -2.677,Y -103.924,Z 270.000,A 0.000,B 0.000,C 180.000,E1 0.000} C_DIS
LIN {X 2.682,Y -103.924,Z 270.000,A 0.000,B 0.000,C 180.000,E1 0.000} C_DIS
LIN {X 8.023,Y -103.649,Z 270.000,A 0.000,B 0.000,C 180.000,E1 0.000} C_DIS
LIN {X 13.349,Y -103.099,Z 270.000,A 0.000,B 0.000,C 180.000,E1 0.000} C_DIS
LIN {X 18.637,Y -102.275,Z 270.000,A 0.000,B 0.000,C 180.000,E1 0.000} C_DIS
LIN {X 23.878,Y -101.180,Z 270.000,A 0.000,B 0.000,C 180.000,E1 0.000} C_DIS
LIN {X 29.054,Y -99.817,Z 270.000,A 0.000,B 0.000,C 180.000,E1 0.000} C_DIS
LIN {X 34.155,Y -98.187,Z 270.000,A 0.000,B 0.000,C 180.000,E1 0.000} C_DIS
LIN {X 39.167,Y -96.299,Z 270.000,A 0.000,B 0.000,C 180.000,E1 0.000} C_DIS
LIN {X 44.070,Y -94.156,Z 270.000,A 0.000,B 0.000,C 180.000,E1 0.000} C_DIS
LIN {X 48.857,Y -91.763,Z 270.000,A 0.000,B 0.000,C 180.000,E1 0.000} C_DIS
LIN {X 53.517,Y -89.126,Z 270.000,A 0.000,B 0.000,C 180.000,E1 0.000} C_DIS
LIN {X 58.033,Y -86.253,Z 270.000,A 0.000,B 0.000,C 180.000,E1 0.000} C_DIS
LIN {X 62.397,Y -83.150,Z 270.000,A 0.000,B 0.000,C 180.000,E1 0.000} C_DIS
LIN {X 66.595,Y -79.828,Z 270.000,A 0.000,B 0.000,C 180.000,E1 0.000} C_DIS
LIN {X 70.617,Y -76.293,Z 270.000,A 0.000,B 0.000,C 180.000,E1 0.000} C_DIS
LIN {X 74.450,Y -72.558,Z 270.000,A 0.000,B 0.000,C 180.000,E1 0.000} C_DIS
LIN {X 78.086,Y -68.629,Z 270.000,A 0.000,B 0.000,C 180.000,E1 0.000} C_DIS
LIN {X 81.517,Y -64.517,Z 270.000,A 0.000,B 0.000,C 180.000,E1 0.000} C_DIS
;rapid-leaky
$VEL.CP=0.3
LIN {X 43.156,Y -74.582,Z 270.000,A 0.000,B 0.000,C 180.000,E1 0.000} C_DIS
;bead-sparse_infill
$VEL.CP=0.21
LIN {X -74.588,Y 43.162,Z 270.000,A 0.000,B 0.000,C 180.000,E1 0.000} C_DIS
;rapid-leaky
$VEL.CP=0.3
LIN {X -94.327,Y 19.712,Z 280.000,A 0.000,B 0.000,C 180.000,E1 0.000} C_DIS
;bead-perimeter_outer
$VEL.CP=0.16
LIN {X -95.216,Y 14.830,Z 280.000,A 0.000,B 0.000,C 180.000,E1 0.000} C_DIS
LIN {X -95.853,Y 9.908,Z 280.000,A 0.000,B 0.000,C 180.000,E1 0.000} C_DIS
LIN {X -96.237,Y 4.960,Z 280.000,A 0.000,B 0.000,C 180.000,E1 0.000} C_DIS
LIN {X -96.365,Y 0.000,Z 280.000,A 0.000,B 0.000,C 180.000,E1 0.000} C_DIS
LIN {X -96.237,Y -4.960,Z 280.000,A 0.000,B 0.000,C 180.000,E1 0.000} C_DIS
LIN {X -95.853,Y -9.908,Z 280.000,A 0.000,B 0.000,C 180.000,E1 0.000} C_DIS
LIN {X -95.216,Y -14.830,Z 280.000,A 0.000,B 0.000,C 180.000,E1 0.000} C_DIS
LIN {X -94.327,Y -19.712,Z 280.000,A 0.000,B 0.000,C 180.000,E1 0.000} C_DIS
LIN {X -93.447,Y -23.441,Z 280.000,A 0.000,B 0.000,C 180.000,E1 0.000} C_DIS
LIN {X -93.188,Y -24.540,Z 280.000,A 0.000,B 0.000,C 180.000,E1 0.000} C_DIS
LIN {X -91.800,Y -29.306,Z 280.000,A 0.000,B 0.000,C 180.000,E1 0.000} C_DIS
LIN {X -90.170,Y -33.993,Z 280.000,A 0.000,B 0.000,C 180.000,E1 0.000} C_DIS
LIN {X -88.301,Y -38.589,Z 280.000,A 0.000,B 0.000,C 180.000,E1 0.000} C_DIS
LIN {X -86.197,Y -43.083,Z 280.000,A 0.000,B 0.000,C 180.000,E1 0.000} C_DIS
LIN {X -83.865,Y -47.464,Z 280.000,A 0.000,B 0.000,C 180.000,E1 0.000} C_DIS
LIN {X -81.310,Y -51.719,Z 280.000,A 0.000,B 0.000,C 180.000,E1 0.000} C_DIS
LIN {X -78.540,Y -55.835,Z 280.000,A 0.000,B 0.000,C 180.000,E1 0.000} C_DIS
LIN {X -75.561,Y -59.805,Z 280.000,A 0.000,B 0.000,C 180.000,E1 0.000} C_DIS
LIN {X -72.383,Y -63.615,Z 280.000,A 0.000,B 0.000,C 180.000,E1 0.000} C_DIS
LIN {X -69.011,Y -67.258,Z 280.000,A 0.000,B 0.000,C 180.000,E1 0.000} C_DIS
LIN {X -65.459,Y -70.721,Z 280.000,A 0.000,B 0.000,C 180.000,E1 0.000} C_DIS
LIN {X -61.730,Y -73.996,Z 280.000,A 0.000,B 0.000,C 180.000,E1 0.000} C_DIS
LIN {X -57.840,Y -77.077,Z 280.000,A 0.000,B 0.000,C 180.000,E1 0.000} C_DIS
LIN {X -53.795,Y -79.951,Z 280.000,A 0.000,B 0.000,C 180.000,E1 0.000} C_DIS
LIN {X -49.607,Y -82.615,Z 280.000,A 0.000,B 0.000,C 180.000,E1 0.000} C_DIS
LIN {X -45.289,Y -85.059,Z 280.000,A 0.000,B 0.000,C 180.000,E1 0.000} C_DIS
LIN {X -40.851,Y -87.278,Z 280.000,A 0.000,B 0.000,C 180.000,E1 0.000} C_DIS
LIN {X -36.303,Y -89.264,Z 280.000,A 0.000,B 0.000,C 180.000,E1 0.000} C_DIS
LIN {X -31.659,Y -91.016,Z 280.000,A 0.000,B 0.000,C 180.000,E1 0.000} C_DIS
LIN {X -26.933,Y -92.525,Z 280.000,A 0.000,B 0.000,C 180.000,E1 0.000} C_DIS
LIN {X -22.135,Y -93.788,Z 280.000,A 0.000,B 0.000,C 180.000,E1 0.000} C_DIS
LIN {X -17.276,Y -94.803,Z 280.000,A 0.000,B 0.000,C 180.000,E1 0.000} C_DIS
LIN {X -12.373,Y -95.567,Z 280.000,A 0.000,B 0.000,C 180.000,E1 0.000} C_DIS
LIN {X -7.437,Y -96.077,Z 280.000,A 0.000,B 0.000,C 180.000,E1 0.000} C_DIS
LIN {X -2.481,Y -96.333,Z 280.000,A 0.000,B 0.000,C 180.000,E1 0.000} C_DIS
LIN {X 2.481,Y -96.333,Z 280.000,A 0.000,B 0.000,C 180.000,E1 0.000} C_DIS
LIN {X 6.310,Y -96.136,Z 280.000,A 0.000,B 0.000,C 180.000,E1 0.000} C_DIS
LIN {X 7.436,Y -96.077,Z 280.000,A 0.000,B 0.000,C 180.000,E1 0.000} C_DIS
LIN {X 12.373,Y -95.567,Z 280.000,A 0.000,B 0.000,C 180.000,E1 0.000} C_DIS
LIN {X 17.276,Y -94.803,Z 280.000,A 0.000,B 0.000,C 180.000,E1 0.000} C_DIS
LIN {X 22.135,Y -93.788,Z 280.000,A 0.000,B 0.000,C 180.000,E1 0.000} C_DIS
LIN {X 26.933,Y -92.525,Z 280.000,A 0.000,B 0.000,C 180.000,E1 0.000} C_DIS
LIN {X 31.659,Y -91.016,Z 280.000,A 0.000,B 0.000,C 180.000,E1 0.000} C_DIS
LIN {X 36.303,Y -89.264,Z 280.000,A 0.000,B 0.000,C 180.000,E1 0.000} C_DIS
LIN {X 40.851,Y -87.278,Z 280.000,A 0.000,B 0.000,C 180.000,E1 0.000} C_DIS
LIN {X 45.289,Y -85.059,Z 280.000,A 0.000,B 0.000,C 180.000,E1 0.000} C_DIS
LIN {X 49.607,Y -82.615,Z 280.000,A 0.000,B 0.000,C 180.000,E1 0.000} C_DIS
LIN {X 53.795,Y -79.951,Z 280.000,A 0.000,B 0.000,C 180.000,E1 0.000} C_DIS
LIN {X 57.840,Y -77.077,Z 280.000,A 0.000,B 0.000,C 180.000,E1 0.000} C_DIS
LIN {X 61.730,Y -73.996,Z 280.000,A 0.000,B 0.000,C 180.000,E1 0.000} C_DIS
LIN {X 65.459,Y -70.721,Z 280.000,A 0.000,B 0.000,C 180.000,E1 0.000} C_DIS
LIN {X 69.011,Y -67.258,Z 280.000,A 0.000,B 0.000,C 180.000,E1 0.000} C_DIS
LIN {X 72.383,Y -63.615,Z 280.000,A 0.000,B 0.000,C 180.000,E1 0.000} C_DIS
LIN {X 75.561,Y -59.805,Z 280.000,A 0.000,B 0.000,C 180.000,E1 0.000} C_DIS
LIN {X 78.540,Y -55.835,Z 280.000,A 0.000,B 0.000,C 180.000,E1 0.000} C_DIS
LIN {X 81.310,Y -51.719,Z 280.000,A 0.000,B 0.000,C 180.000,E1 0.000} C_DIS
LIN {X 83.865,Y -47.464,Z 280.000,A 0.000,B 0.000,C 180.000,E1 0.000} C_DIS
LIN {X 86.197,Y -43.083,Z 280.000,A 0.000,B 0.000,C 180.000,E1 0.000} C_DIS
LIN {X 88.301,Y -38.589,Z 280.000,A 0.000,B 0.000,C 180.000,E1 0.000} C_DIS
LIN {X 90.170,Y -33.993,Z 280.000,A 0.000,B 0.000,C 180.000,E1 0.000} C_DIS
LIN {X 91.429,Y -30.374,Z 280.000,A 0.000,B 0.000,C 180.000,E1 0.000} C_DIS
LIN {X 91.800,Y -29.307,Z 280.000,A 0.000,B 0.000,C 180.000,E1 0.000} C_DIS
LIN {X 93.187,Y -24.541,Z 280.000,A 0.000,B 0.000,C 180.000,E1 0.000} C_DIS
LIN {X 94.327,Y -19.712,Z 280.000,A 0.000,B 0.000,C 180.000,E1 0.000} C_DIS
LIN {X 95.216,Y -14.830,Z 280.000,A 0.000,B 0.000,C 180.000,E1 0.000} C_DIS
LIN {X 95.853,Y -9.908,Z 280.000,A 0.000,B 0.000,C 180.000,E1 0.000} C_DIS
LIN {X 96.237,Y -4.960,Z 280.000,A 0.000,B 0.000,C 180.000,E1 0.000} C_DIS
LIN {X 96.365,Y 0.000,Z 280.000,A 0.000,B 0.000,C 180.000,E1 0.000} C_DIS
LIN {X 96.237,Y 4.960,Z 280.000,A 0.000,B 0.000,C 180.000,E1 0.000} C_DIS
LIN {X 95.853,Y 9.908,Z 280.000,A 0.000,B 0.000,C 180.000,E1 0.000} C_DIS
LIN {X 95.216,Y 14.830,Z 280.000,A 0.000,B 0.000,C 180.000,E1 0.000} C_DIS
LIN {X 94.327,Y 19.712,Z 280.000,A 0.000,B 0.000,C 180.000,E1 0.000} C_DIS
LIN {X 93.188,Y 24.540,Z 280.000,A 0.000,B 0.000,C 180.000,E1 0.000} C_DIS
LIN {X 91.800,Y 29.306,Z 280.000,A 0.000,B 0.000,C 180.000,E1 0.000} C_DIS
LIN {X 90.170,Y 33.993,Z 280.000,A 0.000,B 0.000,C 180.000,E1 0.000} C_DIS
LIN {X 88.301,Y 38.589,Z 280.000,A 0.000,B 0.000,C 180.000,E1 0.000} C_DIS
LIN {X 86.197,Y 43.083,Z 280.000,A 0.000,B 0.000,C 180.000,E1 0.000} C_DIS
LIN {X 83.865,Y 47.464,Z 280.000,A 0.000,B 0.000,C 180.000,E1 0.000} C_DIS
LIN {X 81.310,Y 51.719,Z 280.000,A 0.000,B 0.000,C 180.000,E1 0.000} C_DIS
LIN {X 78.540,Y 55.835,Z 280.000,A 0.000,B 0.000,C 180.000,E1 0.000} C_DIS
LIN {X 75.561,Y 59.805,Z 280.000,A 0.000,B 0.000,C 180.000,E1 0.000} C_DIS
LIN {X 72.383,Y 63.615,Z 280.000,A 0.000,B 0.000,C 180.000,E1 0.000} C_DIS
LIN {X 69.011,Y 67.258,Z 280.000,A 0.000,B 0.000,C 180.000,E1 0.000} C_DIS
LIN {X 65.459,Y 70.721,Z 280.000,A 0.000,B 0.000,C 180.000,E1 0.000} C_DIS
LIN {X 61.730,Y 73.996,Z 280.000,A 0.000,B 0.000,C 180.000,E1 0.000} C_DIS
LIN {X 57.840,Y 77.077,Z 280.000,A 0.000,B 0.000,C 180.000,E1 0.000} C_DIS
LIN {X 53.795,Y 79.951,Z 280.000,A 0.000,B 0.000,C 180.000,E1 0.000} C_DIS
LIN {X 49.607,Y 82.615,Z 280.000,A 0.000,B 0.000,C 180.000,E1 0.000} C_DIS
LIN {X 45.289,Y 85.059,Z 280.000,A 0.000,B 0.000,C 180.000,E1 0.000} C_DIS
LIN {X 40.851,Y 87.278,Z 280.000,A 0.000,B 0.000,C 180.000,E1 0.000} C_DIS
LIN {X 36.303,Y 89.264,Z 280.000,A 0.000,B 0.000,C 180.000,E1 0.000} C_DIS
LIN {X 31.659,Y 91.016,Z 280.000,A 0.000,B 0.000,C 180.000,E1 0.000} C_DIS
LIN {X 26.933,Y 92.525,Z 280.000,A 0.000,B 0.000,C 180.000,E1 0.000} C_DIS
LIN {X 22.135,Y 93.788,Z 280.000,A 0.000,B 0.000,C 180.000,E1 0.000} C_DIS
LIN {X 17.276,Y 94.803,Z 280.000,A 0.000,B 0.000,C 180.000,E1 0.000} C_DIS
LIN {X 12.373,Y 95.567,Z 280.000,A 0.000,B 0.000,C 180.000,E1 0.000} C_DIS
LIN {X 7.437,Y 96.077,Z 280.000,A 0.000,B 0.000,C 180.000,E1 0.000} C_DIS
LIN {X 2.481,Y 96.333,Z 280.000,A 0.000,B 0.000,C 180.000,E1 0.000} C_DIS
LIN {X -2.481,Y 96.333,Z 280.000,A 0.000,B 0.000,C 180.000,E1 0.000} C_DIS
LIN {X -6.310,Y 96.136,Z 280.000,A 0.000,B 0.000,C 180.000,E1 0.000} C_DIS
LIN {X -7.436,Y 96.077,Z 280.000,A 0.000,B 0.000,C 180.000,E1 0.000} C_DIS
LIN {X -12.373,Y 95.567,Z 280.000,A 0.000,B 0.000,C 180.000,E1 0.000} C_DIS
LIN {X -17.276,Y 94.803,Z 280.000,A 0.000,B 0.000,C 180.000,E1 0.000} C_DIS
LIN {X -22.135,Y 93.788,Z 280.000,A 0.000,B 0.000,C 180.000,E1 0.000} C_DIS
LIN {X -26.933,Y 92.525,Z 280.000,A 0.000,B 0.000,C 180.000,E1 0.000} C_DIS
LIN {X -31.659,Y 91.016,Z 280.000,A 0.000,B 0.000,C 180.000,E1 0.000} C_DIS
LIN {X -36.303,Y 89.264,Z 280.000,A 0.000,B 0.000,C 180.000,E1 0.000} C_DIS
LIN {X -40.851,Y 87.278,Z 280.000,A 0.000,B 0.000,C 180.000,E1 0.000} C_DIS
LIN {X -45.289,Y 85.059,Z 280.000,A 0.000,B 0.000,C 180.000,E1 0.000} C_DIS
LIN {X -49.607,Y 82.615,Z 280.000,A 0.000,B 0.000,C 180.000,E1 0.000} C_DIS
LIN {X -53.795,Y 79.951,Z 280.000,A 0.000,B 0.000,C 180.000,E1 0.000} C_DIS
LIN {X -57.840,Y 77.077,Z 280.000,A 0.000,B 0.000,C 180.000,E1 0.000} C_DIS
LIN {X -61.730,Y 73.996,Z 280.000,A 0.000,B 0.000,C 180.000,E1 0.000} C_DIS
LIN {X -65.459,Y 70.721,Z 280.000,A 0.000,B 0.000,C 180.000,E1 0.000} C_DIS
LIN {X -69.011,Y 67.258,Z 280.000,A 0.000,B 0.000,C 180.000,E1 0.000} C_DIS
LIN {X -72.383,Y 63.615,Z 280.000,A 0.000,B 0.000,C 180.000,E1 0.000} C_DIS
LIN {X -75.561,Y 59.805,Z 280.000,A 0.000,B 0.000,C 180.000,E1 0.000} C_DIS
LIN {X -78.540,Y 55.835,Z 280.000,A 0.000,B 0.000,C 180.000,E1 0.000} C_DIS
LIN {X -81.310,Y 51.719,Z 280.000,A 0.000,B 0.000,C 180.000,E1 0.000} C_DIS
LIN {X -83.865,Y 47.464,Z 280.000,A 0.000,B 0.000,C 180.000,E1 0.000} C_DIS
LIN {X -86.197,Y 43.083,Z 280.000,A 0.000,B 0.000,C 180.000,E1 0.000} C_DIS
LIN {X -88.301,Y 38.589,Z 280.000,A 0.000,B 0.000,C 180.000,E1 0.000} C_DIS
LIN {X -90.170,Y 33.993,Z 280.000,A 0.000,B 0.000,C 180.000,E1 0.000} C_DIS
LIN {X -91.800,Y 29.307,Z 280.000,A 0.000,B 0.000,C 180.000,E1 0.000} C_DIS
LIN {X -93.187,Y 24.541,Z 280.000,A 0.000,B 0.000,C 180.000,E1 0.000} C_DIS
LIN {X -94.327,Y 19.712,Z 280.000,A 0.000,B 0.000,C 180.000,E1 0.000} C_DIS
;rapid-leaky
$VEL.CP=0.3
LIN {X -79.110,Y 16.533,Z 280.000,A 0.000,B 0.000,C 180.000,E1 0.000} C_DIS
;bead-perimeter_inner
$VEL.CP=0.16
LIN {X -79.856,Y 12.439,Z 280.000,A 0.000,B 0.000,C 180.000,E1 0.000} C_DIS
LIN {X -80.391,Y 8.309,Z 280.000,A 0.000,B 0.000,C 180.000,E1 0.000} C_DIS
LIN {X -80.713,Y 4.158,Z 280.000,A 0.000,B 0.000,C 180.000,E1 0.000} C_DIS
LIN {X -80.820,Y 0.000,Z 280.000,A 0.000,B 0.000,C 180.000,E1 0.000} C_DIS
LIN {X -80.713,Y -4.158,Z 280.000,A 0.000,B 0.000,C 180.000,E1 0.000} C_DIS
LIN {X -80.391,Y -8.309,Z 280.000,A 0.000,B 0.000,C 180.000,E1 0.000} C_DIS
LIN {X -79.856,Y -12.439,Z 280.000,A 0.000,B 0.000,C 180.000,E1 0.000} C_DIS
LIN {X -79.110,Y -16.534,Z 280.000,A 0.000,B 0.000,C 180.000,E1 0.000} C_DIS
LIN {X -78.323,Y -19.869,Z 280.000,A 0.000,B 0.000,C 180.000,E1 0.000} C_DIS
LIN {X -78.156,Y -20.580,Z 280.000,A 0.000,B 0.000,C 180.000,E1 0.000} C_DIS
LIN {X -76.991,Y -24.579,Z 280.000,A 0.000,B 0.000,C 180.000,E1 0.000} C_DIS
LIN {X -75.624,Y -28.509,Z 280.000,A 0.000,B 0.000,C 180.000,E1 0.000} C_DIS
LIN {X -74.057,Y -32.364,Z 280.000,A 0.000,B 0.000,C 180.000,E1 0.000} C_DIS
LIN {X -72.292,Y -36.133,Z 280.000,A 0.000,B 0.000,C 180.000,E1 0.000} C_DIS
LIN {X -70.336,Y -39.808,Z 280.000,A 0.000,B 0.000,C 180.000,E1 0.000} C_DIS
LIN {X -68.193,Y -43.376,Z 280.000,A 0.000,B 0.000,C 180.000,E1 0.000} C_DIS
LIN {X -65.870,Y -46.828,Z 280.000,A 0.000,B 0.000,C 180.000,E1 0.000} C_DIS
LIN {X -63.372,Y -50.157,Z 280.000,A 0.000,B 0.000,C 180.000,E1 0.000} C_DIS
LIN {X -60.706,Y -53.353,Z 280.000,A 0.000,B 0.000,C 180.000,E1 0.000} C_DIS
LIN {X -57.878,Y -56.409,Z 280.000,A 0.000,B 0.000,C 180.000,E1 0.000} C_DIS
LIN {X -54.900,Y -59.312,Z 280.000,A 0.000,B 0.000,C 180.000,E1 0.000} C_DIS
LIN {X -51.773,Y -62.059,Z 280.000,A 0.000,B 0.000,C 180.000,E1 0.000} C_DIS
LIN {X -48.509,Y -64.643,Z 280.000,A 0.000,B 0.000,C 180.000,E1 0.000} C_DIS
LIN {X -45.118,Y -67.053,Z 280.000,A 0.000,B 0.000,C 180.000,E1 0.000} C_DIS
LIN {X -41.604,Y -69.288,Z 280.000,A 0.000,B 0.000,C 180.000,E1 0.000} C_DIS
LIN {X -37.982,Y -71.338,Z 280.000,A 0.000,B 0.000,C 180.000,E1 0.000} C_DIS
LIN {X -34.262,Y -73.198,Z 280.000,A 0.000,B 0.000,C 180.000,E1 0.000} C_DIS
LIN {X -30.447,Y -74.865,Z 280.000,A 0.000,B 0.000,C 180.000,E1 0.000} C_DIS
LIN {X -26.551,Y -76.334,Z 280.000,A 0.000,B 0.000,C 180.000,E1 0.000} C_DIS
LIN {X -22.589,Y -77.599,Z 280.000,A 0.000,B 0.000,C 180.000,E1 0.000} C_DIS
LIN {X -18.565,Y -78.658,Z 280.000,A 0.000,B 0.000,C 180.000,E1 0.000} C_DIS
LIN {X -14.489,Y -79.510,Z 280.000,A 0.000,B 0.000,C 180.000,E1 0.000} C_DIS
LIN {X -10.377,Y -80.151,Z 280.000,A 0.000,B 0.000,C 180.000,E1 0.000} C_DIS
LIN {X -6.237,Y -80.579,Z 280.000,A 0.000,B 0.000,C 180.000,E1 0.000} C_DIS
LIN {X -2.081,Y -80.793,Z 280.000,A 0.000,B 0.000,C 180.000,E1 0.000} C_DIS
LIN {X 2.081,Y -80.793,Z 280.000,A 0.000,B 0.000,C 180.000,E1 0.000} C_DIS
LIN {X 5.508,Y -80.616,Z 280.000,A 0.000,B 0.000,C 180.000,E1 0.000} C_DIS
LIN {X 6.236,Y -80.579,Z 280.000,A 0.000,B 0.000,C 180.000,E1 0.000} C_DIS
LIN {X 10.377,Y -80.151,Z 280.000,A 0.000,B 0.000,C 180.000,E1 0.000} C_DIS
LIN {X 14.489,Y -79.510,Z 280.000,A 0.000,B 0.000,C 180.000,E1 0.000} C_DIS
LIN {X 18.565,Y -78.658,Z 280.000,A 0.000,B 0.000,C 180.000,E1 0.000} C_DIS
LIN {X 22.589,Y -77.599,Z 280.000,A 0.000,B 0.000,C 180.000,E1 0.000} C_DIS
LIN {X 26.551,Y -76.334,Z 280.000,A 0.000,B 0.000,C 180.000,E1 0.000} C_DIS
LIN {X 30.447,Y -74.865,Z 280.000,A 0.000,B 0.000,C 180.000,E1 0.000} C_DIS
LIN {X 34.262,Y -73.198,Z 280.000,A 0.000,B 0.000,C 180.000,E1 0.000} C_DIS
LIN {X 37.982,Y -71.338,Z 280.000,A 0.000,B 0.000,C 180.000,E1 0.000} C_DIS
LIN {X 41.604,Y -69.288,Z 280.000,A 0.000,B 0.000,C 180.000,E1 0.000} C_DIS
LIN {X 45.118,Y -67.053,Z 280.000,A 0.000,B 0.000,C 180.000,E1 0.000} C_DIS
LIN {X 48.509,Y -64.643,Z 280.000,A 0.000,B 0.000,C 180.000,E1 0.000} C_DIS
LIN {X 51.773,Y -62.059,Z 280.000,A 0.000,B 0.000,C 180.000,E1 0.000} C_DIS
LIN {X 54.900,Y -59.312,Z 280.000,A 0.000,B 0.000,C 180.000,E1 0.000} C_DIS
LIN {X 57.878,Y -56.409,Z 280.000,A 0.000,B 0.000,C 180.000,E1 0.000} C_DIS
LIN {X 60.706,Y -53.353,Z 280.000,A 0.000,B 0.000,C 180.000,E1 0.000} C_DIS
LIN {X 63.372,Y -50.157,Z 280.000,A 0.000,B 0.000,C 180.000,E1 0.000} C_DIS
LIN {X 65.870,Y -46.828,Z 280.000,A 0.000,B 0.000,C 180.000,E1 0.000} C_DIS
LIN {X 68.193,Y -43.376,Z 280.000,A 0.000,B 0.000,C 180.000,E1 0.000} C_DIS
LIN {X 70.336,Y -39.808,Z 280.000,A 0.000,B 0.000,C 180.000,E1 0.000} C_DIS
LIN {X 72.292,Y -36.133,Z 280.000,A 0.000,B 0.000,C 180.000,E1 0.000} C_DIS
LIN {X 74.057,Y -32.364,Z 280.000,A 0.000,B 0.000,C 180.000,E1 0.000} C_DIS
LIN {X 75.625,Y -28.509,Z 280.000,A 0.000,B 0.000,C 180.000,E1 0.000} C_DIS
LIN {X 76.752,Y -25.268,Z 280.000,A 0.000,B 0.000,C 180.000,E1 0.000} C_DIS
LIN {X 76.991,Y -24.582,Z 280.000,A 0.000,B 0.000,C 180.000,E1 0.000} C_DIS
LIN {X 78.155,Y -20.582,Z 280.000,A 0.000,B 0.000,C 180.000,E1 0.000} C_DIS
LIN {X 79.110,Y -16.533,Z 280.000,A 0.000,B 0.000,C 180.000,E1 0.000} C_DIS
LIN {X 79.856,Y -12.439,Z 280.000,A 0.000,B 0.000,C 180.000,E1 0.000} C_DIS
LIN {X 80.391,Y -8.309,Z 280.000,A 0.000,B 0.000,C 180.000,E1 0.000} C_DIS
LIN {X 80.713,Y -4.158,Z 280.000,A 0.000,B 0.000,C 180.000,E1 0.000} C_DIS
LIN {X 80.820,Y 0.000,Z 280.000,A 0.000,B 0.000,C 180.000,E1 0.000} C_DIS
LIN {X 80.713,Y 4.158,Z 280.000,A 0.000,B 0.000,C 180.000,E1 0.000} C_DIS
LIN {X 80.391,Y 8.309,Z 280.000,A 0.000,B 0.000,C 180.000,E1 0.000} C_DIS
LIN {X 79.856,Y 12.439,Z 280.000,A 0.000,B 0.000,C 180.000,E1 0.000} C_DIS
LIN {X 79.110,Y 16.534,Z 280.000,A 0.000,B 0.000,C 180.000,E1 0.000} C_DIS
LIN {X 78.156,Y 20.580,Z 280.000,A 0.000,B 0.000,C 180.000,E1 0.000} C_DIS
LIN {X 76.991,Y 24.579,Z 280.000,A 0.000,B 0.000,C 180.000,E1 0.000} C_DIS
LIN {X 75.624,Y 28.509,Z 280.000,A 0.000,B 0.000,C 180.000,E1 0.000} C_DIS
LIN {X 74.057,Y 32.364,Z 280.000,A 0.000,B 0.000,C 180.000,E1 0.000} C_DIS
LIN {X 72.292,Y 36.133,Z 280.000,A 0.000,B 0.000,C 180.000,E1 0.000} C_DIS
LIN {X 70.336,Y 39.808,Z 280.000,A 0.000,B 0.000,C 180.000,E1 0.000} C_DIS
LIN {X 68.193,Y 43.376,Z 280.000,A 0.000,B 0.000,C 180.000,E1 0.000} C_DIS
LIN {X 65.870,Y 46.828,Z 280.000,A 0.000,B 0.000,C 180.000,E1 0.000} C_DIS
LIN {X 63.372,Y 50.157,Z 280.000,A 0.000,B 0.000,C 180.000,E1 0.000} C_DIS
LIN {X 60.706,Y 53.353,Z 280.000,A 0.000,B 0.000,C 180.000,E1 0.000} C_DIS
LIN {X 57.878,Y 56.409,Z 280.000,A 0.000,B 0.000,C 180.000,E1 0.000} C_DIS
LIN {X 54.900,Y 59.312,Z 280.000,A 0.000,B 0.000,C 180.000,E1 0.000} C_DIS
LIN {X 51.773,Y 62.059,Z 280.000,A 0.000,B 0.000,C 180.000,E1 0.000} C_DIS
LIN {X 48.509,Y 64.643,Z 280.000,A 0.000,B 0.000,C 180.000,E1 0.000} C_DIS
LIN {X 45.118,Y 67.053,Z 280.000,A 0.000,B 0.000,C 180.000,E1 0.000} C_DIS
LIN {X 41.604,Y 69.288,Z 280.000,A 0.000,B 0.000,C 180.000,E1 0.000} C_DIS
LIN {X 37.982,Y 71.338,Z 280.000,A 0.000,B 0.000,C 180.000,E1 0.000} C_DIS
LIN {X 34.262,Y 73.198,Z 280.000,A 0.000,B 0.000,C 180.000,E1 0.000} C_DIS
LIN {X 30.447,Y 74.865,Z 280.000,A 0.000,B 0.000,C 180.000,E1 0.000} C_DIS
LIN {X 26.551,Y 76.334,Z 280.000,A 0.000,B 0.000,C 180.000,E1 0.000} C_DIS
LIN {X 22.589,Y 77.599,Z 280.000,A 0.000,B 0.000,C 180.000,E1 0.000} C_DIS
LIN {X 18.565,Y 78.658,Z 280.000,A 0.000,B 0.000,C 180.000,E1 0.000} C_DIS
LIN {X 14.489,Y 79.510,Z 280.000,A 0.000,B 0.000,C 180.000,E1 0.000} C_DIS
LIN {X 10.377,Y 80.151,Z 280.000,A 0.000,B 0.000,C 180.000,E1 0.000} C_DIS
LIN {X 6.237,Y 80.579,Z 280.000,A 0.000,B 0.000,C 180.000,E1 0.000} C_DIS
LIN {X 2.081,Y 80.793,Z 280.000,A 0.000,B 0.000,C 180.000,E1 0.000} C_DIS
LIN {X -2.081,Y 80.793,Z 280.000,A 0.000,B 0.000,C 180.000,E1 0.000} C_DIS
LIN {X -5.508,Y 80.616,Z 280.000,A 0.000,B 0.000,C 180.000,E1 0.000} C_DIS
LIN {X -6.236,Y 80.579,Z 280.000,A 0.000,B 0.000,C 180.000,E1 0.000} C_DIS
LIN {X -10.377,Y 80.151,Z 280.000,A 0.000,B 0.000,C 180.000,E1 0.000} C_DIS
LIN {X -14.489,Y 79.510,Z 280.000,A 0.000,B 0.000,C 180.000,E1 0.000} C_DIS
LIN {X -18.565,Y 78.658,Z 280.000,A 0.000,B 0.000,C 180.000,E1 0.000} C_DIS
LIN {X -22.589,Y 77.599,Z 280.000,A 0.000,B 0.000,C 180.000,E1 0.000} C_DIS
LIN {X -26.551,Y 76.334,Z 280.000,A 0.000,B 0.000,C 180.000,E1 0.000} C_DIS
LIN {X -30.447,Y 74.865,Z 280.000,A 0.000,B 0.000,C 180.000,E1 0.000} C_DIS
LIN {X -34.262,Y 73.198,Z 280.000,A 0.000,B 0.000,C 180.000,E1 0.000} C_DIS
LIN {X -37.982,Y 71.338,Z 280.000,A 0.000,B 0.000,C 180.000,E1 0.000} C_DIS
LIN {X -41.604,Y 69.288,Z 280.000,A 0.000,B 0.000,C 180.000,E1 0.000} C_DIS
LIN {X -45.118,Y 67.053,Z 280.000,A 0.000,B 0.000,C 180.000,E1 0.000} C_DIS
LIN {X -48.509,Y 64.643,Z 280.000,A 0.000,B 0.000,C 180.000,E1 0.000} C_DIS
LIN {X -51.773,Y 62.059,Z 280.000,A 0.000,B 0.000,C 180.000,E1 0.000} C_DIS
LIN {X -54.900,Y 59.312,Z 280.000,A 0.000,B 0.000,C 180.000,E1 0.000} C_DIS
LIN {X -57.878,Y 56.409,Z 280.000,A 0.000,B 0.000,C 180.000,E1 0.000} C_DIS
LIN {X -60.706,Y 53.353,Z 280.000,A 0.000,B 0.000,C 180.000,E1 0.000} C_DIS
LIN {X -63.372,Y 50.157,Z 280.000,A 0.000,B 0.000,C 180.000,E1 0.000} C_DIS
LIN {X -65.870,Y 46.828,Z 280.000,A 0.000,B 0.000,C 180.000,E1 0.000} C_DIS
LIN {X -68.193,Y 43.376,Z 280.000,A 0.000,B 0.000,C 180.000,E1 0.000} C_DIS
LIN {X -70.336,Y 39.808,Z 280.000,A 0.000,B 0.000,C 180.000,E1 0.000} C_DIS
LIN {X -72.292,Y 36.133,Z 280.000,A 0.000,B 0.000,C 180.000,E1 0.000} C_DIS
LIN {X -74.057,Y 32.364,Z 280.000,A 0.000,B 0.000,C 180.000,E1 0.000} C_DIS
LIN {X -75.625,Y 28.509,Z 280.000,A 0.000,B 0.000,C 180.000,E1 0.000} C_DIS
LIN {X -76.991,Y 24.582,Z 280.000,A 0.000,B 0.000,C 180.000,E1 0.000} C_DIS
LIN {X -78.155,Y 20.582,Z 280.000,A 0.000,B 0.000,C 180.000,E1 0.000} C_DIS
LIN {X -79.110,Y 16.533,Z 280.000,A 0.000,B 0.000,C 180.000,E1 0.000} C_DIS
;rapid-leaky
$VEL.CP=0.3
LIN {X -57.426,Y -26.000,Z 280.000,A 0.000,B 0.000,C 180.000,E1 0.000} C_DIS
;bead-sparse_infill
$VEL.CP=0.16
LIN {X 26.000,Y 57.426,Z 280.000,A 0.000,B 0.000,C 180.000,E1 0.000} C_DIS
$VEL.CP=0.3
LIN {X 26.000,Y 57.426,Z 280.000,A 0.000,B 0.000,C 180.000,E1 0.000} C_DIS
EXTRUDER_STATE=FALSE

LIN {X -301.078,Y -172.834,Z 690.000,A 0.000,B 0.000,C 180.000,E1 0.000} C_DIS
LIN {X -65.136,Y -6.733,Z 690.000,A 0.000,B 0.000,C 180.000,E1 0.000} C_DIS
LIN {X -65.136,Y -6.733,Z 290.000,A 0.000,B 0.000,C 180.000,E1 0.000} C_DIS
LIN {X -65.136,Y -6.733,Z 290.000,A 0.000,B 0.000,C 180.000,E1 0.000} C_DIS
EXTRUDER_STATE=TRUE

;bead-perimeter_outer
$VEL.CP=0.16
LIN {X -64.703,Y -10.078,Z 290.000,A 0.000,B 0.000,C 180.000,E1 0.000} C_DIS
LIN {X -64.099,Y -13.394,Z 290.000,A 0.000,B 0.000,C 180.000,E1 0.000} C_DIS
LIN {X -63.324,Y -16.676,Z 290.000,A 0.000,B 0.000,C 180.000,E1 0.000} C_DIS
LIN {X -62.382,Y -19.914,Z 290.000,A 0.000,B 0.000,C 180.000,E1 0.000} C_DIS
LIN {X -61.274,Y -23.098,Z 290.000,A 0.000,B 0.000,C 180.000,E1 0.000} C_DIS
LIN {X -60.003,Y -26.224,Z 290.000,A 0.000,B 0.000,C 180.000,E1 0.000} C_DIS
LIN {X -58.574,Y -29.278,Z 290.000,A 0.000,B 0.000,C 180.000,E1 0.000} C_DIS
LIN {X -56.990,Y -32.252,Z 290.000,A 0.000,B 0.000,C 180.000,E1 0.000} C_DIS
LIN {X -55.253,Y -35.144,Z 290.000,A 0.000,B 0.000,C 180.000,E1 0.000} C_DIS
LIN {X -53.371,Y -37.942,Z 290.000,A 0.000,B 0.000,C 180.000,E1 0.000} C_DIS
LIN {X -51.346,Y -40.640,Z 290.000,A 0.000,B 0.000,C 180.000,E1 0.000} C_DIS
LIN {X -49.186,Y -43.230,Z 290.000,A 0.000,B 0.000,C 180.000,E1 0.000} C_DIS
LIN {X -46.898,Y -45.702,Z 290.000,A 0.000,B 0.000,C 180.000,E1 0.000} C_DIS
LIN {X -44.480,Y -48.058,Z 290.000,A 0.000,B 0.000,C 180.000,E1 0.000} C_DIS
LIN {X -41.948,Y -50.285,Z 290.000,A 0.000,B 0.000,C 180.000,E1 0.000} C_DIS
LIN {X -39.304,Y -52.377,Z 290.000,A 0.000,B 0.000,C 180.000,E1 0.000} C_DIS
LIN {X -36.558,Y -54.330,Z 290.000,A 0.000,B 0.000,C 180.000,E1 0.000} C_DIS
LIN {X -33.710,Y -56.140,Z 290.000,A 0.000,B 0.000,C 180.000,E1 0.000} C_DIS
LIN {X -30.782,Y -57.798,Z 290.000,A 0.000,B 0.000,C 180.000,E1 0.000} C_DIS
LIN {X -27.760,Y -59.309,Z 290.000,A 0.000,B 0.000,C 180.000,E1 0.000} C_DIS
LIN {X -24.670,Y -60.659,Z 290.000,A 0.000,B 0.000,C 180.000,E1 0.000} C_DIS
LIN {X -21.515,Y -61.848,Z 290.000,A 0.000,B 0.000,C 180.000,E1 0.000} C_DIS
LIN {X -18.301,Y -62.874,Z 290.000,A 0.000,B 0.000,C 180.000,E1 0.000} C_DIS
LIN {X -15.042,Y -63.733,Z 290.000,A 0.000,B 0.000,C 180.000,E1 0.000} C_DIS
LIN {X -11.741,Y -64.422,Z 290.000,A 0.000,B 0.000,C 180.000,E1 0.000} C_DIS
LIN {X -8.408,Y -64.941,Z 290.000,A 0.000,B 0.000,C 180.000,E1 0.000} C_DIS
LIN {X -5.053,Y -65.288,Z 290.000,A 0.000,B 0.000,C 180.000,E1 0.000} C_DIS
LIN {X -1.686,Y -65.462,Z 290.000,A 0.000,B 0.000,C 180.000,E1 0.000} C_DIS
LIN {X 1.686,Y -65.462,Z 290.000,A 0.000,B 0.000,C 180.000,E1 0.000} C_DIS
LIN {X 5.053,Y -65.288,Z 290.000,A 0.000,B 0.000,C 180.000,E1 0.000} C_DIS
LIN {X 8.408,Y -64.941,Z 290.000,A 0.000,B 0.000,C 180.000,E1 0.000} C_DIS
LIN {X 11.741,Y -64.422,Z 290.000,A 0.000,B 0.000,C 180.000,E1 0.000} C_DIS
LIN {X 15.042,Y -63.733,Z 290.000,A 0.000,B 0.000,C 180.000,E1 0.000} C_DIS
LIN {X 18.301,Y -62.874,Z 290.000,A 0.000,B 0.000,C 180.000,E1 0.000} C_DIS
LIN {X 21.515,Y -61.848,Z 290.000,A 0.000,B 0.000,C 180.000,E1 0.000} C_DIS
LIN {X 24.670,Y -60.659,Z 290.000,A 0.000,B 0.000,C 180.000,E1 0.000} C_DIS
LIN {X 27.760,Y -59.309,Z 290.000,A 0.000,B 0.000,C 180.000,E1 0.000} C_DIS
LIN {X 30.774,Y -57.802,Z 290.000,A 0.000,B 0.000,C 180.000,E1 0.000} C_DIS
LIN {X 33.711,Y -56.139,Z 290.000,A 0.000,B 0.000,C 180.000,E1 0.000} C_DIS
LIN {X 36.558,Y -54.330,Z 290.000,A 0.000,B 0.000,C 180.000,E1 0.000} C_DIS
LIN {X 39.304,Y -52.377,Z 290.000,A 0.000,B 0.000,C 180.000,E1 0.000} C_DIS
LIN {X 41.948,Y -50.285,Z 290.000,A 0.000,B 0.000,C 180.000,E1 0.000} C_DIS
LIN {X 44.480,Y -48.058,Z 290.000,A 0.000,B 0.000,C 180.000,E1 0.000} C_DIS
LIN {X 46.898,Y -45.702,Z 290.000,A 0.000,B 0.000,C 180.000,E1 0.000} C_DIS
LIN {X 49.186,Y -43.230,Z 290.000,A 0.000,B 0.000,C 180.000,E1 0.000} C_DIS
LIN {X 51.346,Y -40.640,Z 290.000,A 0.000,B 0.000,C 180.000,E1 0.000} C_DIS
LIN {X 53.371,Y -37.942,Z 290.000,A 0.000,B 0.000,C 180.000,E1 0.000} C_DIS
LIN {X 55.253,Y -35.144,Z 290.000,A 0.000,B 0.000,C 180.000,E1 0.000} C_DIS
LIN {X 56.990,Y -32.252,Z 290.000,A 0.000,B 0.000,C 180.000,E1 0.000} C_DIS
LIN {X 58.574,Y -29.278,Z 290.000,A 0.000,B 0.000,C 180.000,E1 0.000} C_DIS
LIN {X 60.003,Y -26.224,Z 290.000,A 0.000,B 0.000,C 180.000,E1 0.000} C_DIS
LIN {X 61.274,Y -23.098,Z 290.000,A 0.000,B 0.000,C 180.000,E1 0.000} C_DIS
LIN {X 62.382,Y -19.914,Z 290.000,A 0.000,B 0.000,C 180.000,E1 0.000} C_DIS
LIN {X 63.324,Y -16.676,Z 290.000,A 0.000,B 0.000,C 180.000,E1 0.000} C_DIS
LIN {X 64.099,Y -13.394,Z 290.000,A 0.000,B 0.000,C 180.000,E1 0.000} C_DIS
LIN {X 64.704,Y -10.077,Z 290.000,A 0.000,B 0.000,C 180.000,E1 0.000} C_DIS
LIN {X 65.136,Y -6.740,Z 290.000,A 0.000,B 0.000,C 180.000,E1 0.000} C_DIS
LIN {X 65.397,Y -3.370,Z 290.000,A 0.000,B 0.000,C 180.000,E1 0.000} C_DIS
LIN {X 65.484,Y 0.000,Z 290.000,A 0.000,B 0.000,C 180.000,E1 0.000} C_DIS
LIN {X 65.397,Y 3.370,Z 290.000,A 0.000,B 0.000,C 180.000,E1 0.000} C_DIS
LIN {X 65.136,Y 6.733,Z 290.000,A 0.000,B 0.000,C 180.000,E1 0.000} C_DIS
LIN {X 64.703,Y 10.078,Z 290.000,A 0.000,B 0.000,C 180.000,E1 0.000} C_DIS
LIN {X 64.099,Y 13.394,Z 290.000,A 0.000,B 0.000,C 180.000,E1 0.000} C_DIS
LIN {X 63.324,Y 16.676,Z 290.000,A 0.000,B 0.000,C 180.000,E1 0.000} C_DIS
LIN {X 62.382,Y 19.914,Z 290.000,A 0.000,B 0.000,C 180.000,E1 0.000} C_DIS
LIN {X 61.274,Y 23.098,Z 290.000,A 0.000,B 0.000,C 180.000,E1 0.000} C_DIS
LIN {X 60.003,Y 26.224,Z 290.000,A 0.000,B 0.000,C 180.000,E1 0.000} C_DIS
LIN {X 58.574,Y 29.278,Z 290.000,A 0.000,B 0.000,C 180.000,E1 0.000} C_DIS
LIN {X 56.990,Y 32.252,Z 290.000,A 0.000,B 0.000,C 180.000,E1 0.000} C_DIS
LIN {X 55.253,Y 35.144,Z 290.000,A 0.000,B 0.000,C 180.000,E1 0.000} C_DIS
LIN {X 53.371,Y 37.942,Z 290.000,A 0.000,B 0.000,C 180.000,E1 0.000} C_DIS
LIN {X 51.346,Y 40.640,Z 290.000,A 0.000,B 0.000,C 180.000,E1 0.000} C_DIS
LIN {X 49.186,Y 43.230,Z 290.000,A 0.000,B 0.000,C 180.000,E1 0.000} C_DIS
LIN {X 46.898,Y 45.702,Z 290.000,A 0.000,B 0.000,C 180.000,E1 0.000} C_DIS
LIN {X 44.480,Y 48.058,Z 290.000,A 0.000,B 0.000,C 180.000,E1 0.000} C_DIS
LIN {X 41.948,Y 50.285,Z 290.000,A 0.000,B 0.000,C 180.000,E1 0.000} C_DIS
LIN {X 39.304,Y 52.377,Z 290.000,A 0.000,B 0.000,C 180.000,E1 0.000} C_DIS
LIN {X 36.558,Y 54.330,Z 290.000,A 0.000,B 0.000,C 180.000,E1 0.000} C_DIS
LIN {X 33.710,Y 56.140,Z 290.000,A 0.000,B 0.000,C 180.000,E1 0.000} C_DIS
LIN {X 30.782,Y 57.798,Z 290.000,A 0.000,B 0.000,C 180.000,E1 0.000} C_DIS
LIN {X 27.760,Y 59.309,Z 290.000,A 0.000,B 0.000,C 180.000,E1 0.000} C_DIS
LIN {X 24.670,Y 60.659,Z 290.000,A 0.000,B 0.000,C 180.000,E1 0.000} C_DIS
LIN {X 21.515,Y 61.848,Z 290.000,A 0.000,B 0.000,C 180.000,E1 0.000} C_DIS
LIN {X 18.301,Y 62.874,Z 290.000,A 0.000,B 0.000,C 180.000,E1 0.000} C_DIS
LIN {X 15.042,Y 63.733,Z 290.000,A 0.000,B 0.000,C 180.000,E1 0.000} C_DIS
LIN {X 11.741,Y 64.422,Z 290.000,A 0.000,B 0.000,C 180.000,E1 0.000} C_DIS
LIN {X 8.408,Y 64.941,Z 290.000,A 0.000,B 0.000,C 180.000,E1 0.000} C_DIS
LIN {X 5.053,Y 65.288,Z 290.000,A 0.000,B 0.000,C 180.000,E1 0.000} C_DIS
LIN {X 1.686,Y 65.462,Z 290.000,A 0.000,B 0.000,C 180.000,E1 0.000} C_DIS
LIN {X -1.686,Y 65.462,Z 290.000,A 0.000,B 0.000,C 180.000,E1 0.000} C_DIS
LIN {X -5.053,Y 65.288,Z 290.000,A 0.000,B 0.000,C 180.000,E1 0.000} C_DIS
LIN {X -8.408,Y 64.941,Z 290.000,A 0.000,B 0.000,C 180.000,E1 0.000} C_DIS
LIN {X -11.741,Y 64.422,Z 290.000,A 0.000,B 0.000,C 180.000,E1 0.000} C_DIS
LIN {X -15.042,Y 63.733,Z 290.000,A 0.000,B 0.000,C 180.000,E1 0.000} C_DIS
LIN {X -18.301,Y 62.874,Z 290.000,A 0.000,B 0.000,C 180.000,E1 0.000} C_DIS
LIN {X -21.515,Y 61.848,Z 290.000,A 0.000,B 0.000,C 180.000,E1 0.000} C_DIS
LIN {X -24.670,Y 60.659,Z 290.000,A 0.000,B 0.000,C 180.000,E1 0.000} C_DIS
LIN {X -27.760,Y 59.309,Z 290.000,A 0.000,B 0.000,C 180.000,E1 0.000} C_DIS
LIN {X -30.774,Y 57.802,Z 290.000,A 0.000,B 0.000,C 180.000,E1 0.000} C_DIS
LIN {X -33.711,Y 56.139,Z 290.000,A 0.000,B 0.000,C 180.000,E1 0.000} C_DIS
LIN {X -36.558,Y 54.330,Z 290.000,A 0.000,B 0.000,C 180.000,E1 0.000} C_DIS
LIN {X -39.304,Y 52.377,Z 290.000,A 0.000,B 0.000,C 180.000,E1 0.000} C_DIS
LIN {X -41.948,Y 50.285,Z 290.000,A 0.000,B 0.000,C 180.000,E1 0.000} C_DIS
LIN {X -44.480,Y 48.058,Z 290.000,A 0.000,B 0.000,C 180.000,E1 0.000} C_DIS
LIN {X -46.898,Y 45.702,Z 290.000,A 0.000,B 0.000,C 180.000,E1 0.000} C_DIS
LIN {X -49.186,Y 43.230,Z 290.000,A 0.000,B 0.000,C 180.000,E1 0.000} C_DIS
LIN {X -51.346,Y 40.640,Z 290.000,A 0.000,B 0.000,C 180.000,E1 0.000} C_DIS
LIN {X -53.371,Y 37.942,Z 290.000,A 0.000,B 0.000,C 180.000,E1 0.000} C_DIS
LIN {X -55.253,Y 35.144,Z 290.000,A 0.000,B 0.000,C 180.000,E1 0.000} C_DIS
LIN {X -56.990,Y 32.252,Z 290.000,A 0.000,B 0.000,C 180.000,E1 0.000} C_DIS
LIN {X -58.574,Y 29.278,Z 290.000,A 0.000,B 0.000,C 180.000,E1 0.000} C_DIS
LIN {X -60.003,Y 26.224,Z 290.000,A 0.000,B 0.000,C 180.000,E1 0.000} C_DIS
LIN {X -61.274,Y 23.098,Z 290.000,A 0.000,B 0.000,C 180.000,E1 0.000} C_DIS
LIN {X -62.382,Y 19.914,Z 290.000,A 0.000,B 0.000,C 180.000,E1 0.000} C_DIS
LIN {X -63.324,Y 16.676,Z 290.000,A 0.000,B 0.000,C 180.000,E1 0.000} C_DIS
LIN {X -64.099,Y 13.394,Z 290.000,A 0.000,B 0.000,C 180.000,E1 0.000} C_DIS
LIN {X -64.704,Y 10.077,Z 290.000,A 0.000,B 0.000,C 180.000,E1 0.000} C_DIS
LIN {X -65.136,Y 6.740,Z 290.000,A 0.000,B 0.000,C 180.000,E1 0.000} C_DIS
LIN {X -65.397,Y 3.370,Z 290.000,A 0.000,B 0.000,C 180.000,E1 0.000} C_DIS
LIN {X -65.484,Y 0.000,Z 290.000,A 0.000,B 0.000,C 180.000,E1 0.000} C_DIS
LIN {X -65.397,Y -3.370,Z 290.000,A 0.000,B 0.000,C 180.000,E1 0.000} C_DIS
LIN {X -65.136,Y -6.733,Z 290.000,A 0.000,B 0.000,C 180.000,E1 0.000} C_DIS
;rapid-leaky
$VEL.CP=0.3
LIN {X -49.674,Y -5.134,Z 290.000,A 0.000,B 0.000,C 180.000,E1 0.000} C_DIS
;bead-perimeter_inner
$VEL.CP=0.16
LIN {X -49.343,Y -7.686,Z 290.000,A 0.000,B 0.000,C 180.000,E1 0.000} C_DIS
LIN {X -48.883,Y -10.214,Z 290.000,A 0.000,B 0.000,C 180.000,E1 0.000} C_DIS
LIN {X -48.292,Y -12.718,Z 290.000,A 0.000,B 0.000,C 180.000,E1 0.000} C_DIS
LIN {X -47.573,Y -15.187,Z 290.000,A 0.000,B 0.000,C 180.000,E1 0.000} C_DIS
LIN {X -46.729,Y -17.614,Z 290.000,A 0.000,B 0.000,C 180.000,E1 0.000} C_DIS
LIN {X -45.758,Y -20.000,Z 290.000,A 0.000,B 0.000,C 180.000,E1 0.000} C_DIS
LIN {X -44.669,Y -22.330,Z 290.000,A 0.000,B 0.000,C 180.000,E1 0.000} C_DIS
LIN {X -43.463,Y -24.594,Z 290.000,A 0.000,B 0.000,C 180.000,E1 0.000} C_DIS
LIN {X -42.137,Y -26.801,Z 290.000,A 0.000,B 0.000,C 180.000,E1 0.000} C_DIS
LIN {X -40.701,Y -28.935,Z 290.000,A 0.000,B 0.000,C 180.000,E1 0.000} C_DIS
LIN {X -39.156,Y -30.993,Z 290.000,A 0.000,B 0.000,C 180.000,E1 0.000} C_DIS
LIN {X -37.509,Y -32.969,Z 290.000,A 0.000,B 0.000,C 180.000,E1 0.000} C_DIS
LIN {X -35.767,Y -34.851,Z 290.000,A 0.000,B 0.000,C 180.000,E1 0.000} C_DIS
LIN {X -33.920,Y -36.650,Z 290.000,A 0.000,B 0.000,C 180.000,E1 0.000} C_DIS
LIN {X -31.988,Y -38.349,Z 290.000,A 0.000,B 0.000,C 180.000,E1 0.000} C_DIS
LIN {X -29.974,Y -39.943,Z 290.000,A 0.000,B 0.000,C 180.000,E1 0.000} C_DIS
LIN {X -27.882,Y -41.431,Z 290.000,A 0.000,B 0.000,C 180.000,E1 0.000} C_DIS
LIN {X -25.707,Y -42.813,Z 290.000,A 0.000,B 0.000,C 180.000,E1 0.000} C_DIS
LIN {X -23.477,Y -44.076,Z 290.000,A 0.000,B 0.000,C 180.000,E1 0.000} C_DIS
LIN {X -21.170,Y -45.230,Z 290.000,A 0.000,B 0.000,C 180.000,E1 0.000} C_DIS
LIN {X -18.815,Y -46.259,Z 290.000,A 0.000,B 0.000,C 180.000,E1 0.000} C_DIS
LIN {X -16.408,Y -47.166,Z 290.000,A 0.000,B 0.000,C 180.000,E1 0.000} C_DIS
LIN {X -13.956,Y -47.949,Z 290.000,A 0.000,B 0.000,C 180.000,E1 0.000} C_DIS
LIN {X -11.471,Y -48.603,Z 290.000,A 0.000,B 0.000,C 180.000,E1 0.000} C_DIS
LIN {X -8.956,Y -49.129,Z 290.000,A 0.000,B 0.000,C 180.000,E1 0.000} C_DIS
LIN {X -6.411,Y -49.525,Z 290.000,A 0.000,B 0.000,C 180.000,E1 0.000} C_DIS
LIN {X -3.852,Y -49.790,Z 290.000,A 0.000,B 0.000,C 180.000,E1 0.000} C_DIS
LIN {X -1.286,Y -49.922,Z 290.000,A 0.000,B 0.000,C 180.000,E1 0.000} C_DIS
LIN {X 1.286,Y -49.922,Z 290.000,A 0.000,B 0.000,C 180.000,E1 0.000} C_DIS
LIN {X 3.852,Y -49.790,Z 290.000,A 0.000,B 0.000,C 180.000,E1 0.000} C_DIS
LIN {X 6.411,Y -49.525,Z 290.000,A 0.000,B 0.000,C 180.000,E1 0.000} C_DIS
LIN {X 8.956,Y -49.129,Z 290.000,A 0.000,B 0.000,C 180.000,E1 0.000} C_DIS
LIN {X 11.471,Y -48.603,Z 290.000,A 0.000,B 0.000,C 180.000,E1 0.000} C_DIS
LIN {X 13.956,Y -47.949,Z 290.000,A 0.000,B 0.000,C 180.000,E1 0.000} C_DIS
LIN {X 16.408,Y -47.166,Z 290.000,A 0.000,B 0.000,C 180.000,E1 0.000} C_DIS
LIN {X 18.815,Y -46.259,Z 290.000,A 0.000,B 0.000,C 180.000,E1 0.000} C_DIS
LIN {X 21.170,Y -45.230,Z 290.000,A 0.000,B 0.000,C 180.000,E1 0.000} C_DIS
LIN {X 23.465,Y -44.082,Z 290.000,A 0.000,B 0.000,C 180.000,E1 0.000} C_DIS
LIN {X 25.709,Y -42.812,Z 290.000,A 0.000,B 0.000,C 180.000,E1 0.000} C_DIS
LIN {X 27.882,Y -41.431,Z 290.000,A 0.000,B 0.000,C 180.000,E1 0.000} C_DIS
LIN {X 29.974,Y -39.943,Z 290.000,A 0.000,B 0.000,C 180.000,E1 0.000} C_DIS
LIN {X 31.988,Y -38.349,Z 290.000,A 0.000,B 0.000,C 180.000,E1 0.000} C_DIS
LIN {X 33.920,Y -36.650,Z 290.000,A 0.000,B 0.000,C 180.000,E1 0.000} C_DIS
LIN {X 35.767,Y -34.851,Z 290.000,A 0.000,B 0.000,C 180.000,E1 0.000} C_DIS
LIN {X 37.509,Y -32.969,Z 290.000,A 0.000,B 0.000,C 180.000,E1 0.000} C_DIS
LIN {X 39.156,Y -30.993,Z 290.000,A 0.000,B 0.000,C 180.000,E1 0.000} C_DIS
LIN {X 40.701,Y -28.935,Z 290.000,A 0.000,B 0.000,C 180.000,E1 0.000} C_DIS
LIN {X 42.137,Y -26.801,Z 290.000,A 0.000,B 0.000,C 180.000,E1 0.000} C_DIS
LIN {X 43.463,Y -24.594,Z 290.000,A 0.000,B 0.000,C 180.000,E1 0.000} C_DIS
LIN {X 44.669,Y -22.330,Z 290.000,A 0.000,B 0.000,C 180.000,E1 0.000} C_DIS
LIN {X 45.758,Y -20.000,Z 290.000,A 0.000,B 0.000,C 180.000,E1 0.000} C_DIS
LIN {X 46.729,Y -17.614,Z 290.000,A 0.000,B 0.000,C 180.000,E1 0.000} C_DIS
LIN {X 47.573,Y -15.187,Z 290.000,A 0.000,B 0.000,C 180.000,E1 0.000} C_DIS
LIN {X 48.292,Y -12.718,Z 290.000,A 0.000,B 0.000,C 180.000,E1 0.000} C_DIS
LIN {X 48.883,Y -10.214,Z 290.000,A 0.000,B 0.000,C 180.000,E1 0.000} C_DIS
LIN {X 49.344,Y -7.684,Z 290.000,A 0.000,B 0.000,C 180.000,E1 0.000} C_DIS
LIN {X 49.673,Y -5.144,Z 290.000,A 0.000,B 0.000,C 180.000,E1 0.000} C_DIS
LIN {X 49.873,Y -2.567,Z 290.000,A 0.000,B 0.000,C 180.000,E1 0.000} C_DIS
LIN {X 49.939,Y 0.000,Z 290.000,A 0.000,B 0.000,C 180.000,E1 0.000} C_DIS
LIN {X 49.873,Y 2.567,Z 290.000,A 0.000,B 0.000,C 180.000,E1 0.000} C_DIS
LIN {X 49.674,Y 5.134,Z 290.000,A 0.000,B 0.000,C 180.000,E1 0.000} C_DIS
LIN {X 49.343,Y 7.686,Z 290.000,A 0.000,B 0.000,C 180.000,E1 0.000} C_DIS
LIN {X 48.883,Y 10.214,Z 290.000,A 0.000,B 0.000,C 180.000,E1 0.000} C_DIS
LIN {X 48.292,Y 12.718,Z 290.000,A 0.000,B 0.000,C 180.000,E1 0.000} C_DIS
LIN {X 47.573,Y 15.187,Z 290.000,A 0.000,B 0.000,C 180.000,E1 0.000} C_DIS
LIN {X 46.729,Y 17.614,Z 290.000,A 0.000,B 0.000,C 180.000,E1 0.000} C_DIS
LIN {X 45.758,Y 20.000,Z 290.000,A 0.000,B 0.000,C 180.000,E1 0.000} C_DIS
LIN {X 44.669,Y 22.330,Z 290.000,A 0.000,B 0.000,C 180.000,E1 0.000} C_DIS
LIN {X 43.463,Y 24.594,Z 290.000,A 0.000,B 0.000,C 180.000,E1 0.000} C_DIS
LIN {X 42.137,Y 26.801,Z 290.000,A 0.000,B 0.000,C 180.000,E1 0.000} C_DIS
LIN {X 40.701,Y 28.935,Z 290.000,A 0.000,B 0.000,C 180.000,E1 0.000} C_DIS
LIN {X 39.156,Y 30.993,Z 290.000,A 0.000,B 0.000,C 180.000,E1 0.000} C_DIS
LIN {X 37.509,Y 32.969,Z 290.000,A 0.000,B 0.000,C 180.000,E1 0.000} C_DIS
LIN {X 35.767,Y 34.851,Z 290.000,A 0.000,B 0.000,C 180.000,E1 0.000} C_DIS
LIN {X 33.920,Y 36.650,Z 290.000,A 0.000,B 0.000,C 180.000,E1 0.000} C_DIS
LIN {X 31.988,Y 38.349,Z 290.000,A 0.000,B 0.000,C 180.000,E1 0.000} C_DIS
LIN {X 29.974,Y 39.943,Z 290.000,A 0.000,B 0.000,C 180.000,E1 0.000} C_DIS
LIN {X 27.882,Y 41.431,Z 290.000,A 0.000,B 0.000,C 180.000,E1 0.000} C_DIS
LIN {X 25.707,Y 42.813,Z 290.000,A 0.000,B 0.000,C 180.000,E1 0.000} C_DIS
LIN {X 23.477,Y 44.076,Z 290.000,A 0.000,B 0.000,C 180.000,E1 0.000} C_DIS
LIN {X 21.170,Y 45.230,Z 290.000,A 0.000,B 0.000,C 180.000,E1 0.000} C_DIS
LIN {X 18.815,Y 46.259,Z 290.000,A 0.000,B 0.000,C 180.000,E1 0.000} C_DIS
LIN {X 16.408,Y 47.166,Z 290.000,A 0.000,B 0.000,C 180.000,E1 0.000} C_DIS
LIN {X 13.956,Y 47.949,Z 290.000,A 0.000,B 0.000,C 180.000,E1 0.000} C_DIS
LIN {X 11.471,Y 48.603,Z 290.000,A 0.000,B 0.000,C 180.000,E1 0.000} C_DIS
LIN {X 8.956,Y 49.129,Z 290.000,A 0.000,B 0.000,C 180.000,E1 0.000} C_DIS
LIN {X 6.411,Y 49.525,Z 290.000,A 0.000,B 0.000,C 180.000,E1 0.000} C_DIS
LIN {X 3.852,Y 49.790,Z 290.000,A 0.000,B 0.000,C 180.000,E1 0.000} C_DIS
LIN {X 1.286,Y 49.922,Z 290.000,A 0.000,B 0.000,C 180.000,E1 0.000} C_DIS
LIN {X -1.286,Y 49.922,Z 290.000,A 0.000,B 0.000,C 180.000,E1 0.000} C_DIS
LIN {X -3.852,Y 49.790,Z 290.000,A 0.000,B 0.000,C 180.000,E1 0.000} C_DIS
LIN {X -6.411,Y 49.525,Z 290.000,A 0.000,B 0.000,C 180.000,E1 0.000} C_DIS
LIN {X -8.956,Y 49.129,Z 290.000,A 0.000,B 0.000,C 180.000,E1 0.000} C_DIS
LIN {X -11.471,Y 48.603,Z 290.000,A 0.000,B 0.000,C 180.000,E1 0.000} C_DIS
LIN {X -13.956,Y 47.949,Z 290.000,A 0.000,B 0.000,C 180.000,E1 0.000} C_DIS
LIN {X -16.408,Y 47.166,Z 290.000,A 0.000,B 0.000,C 180.000,E1 0.000} C_DIS
LIN {X -18.815,Y 46.259,Z 290.000,A 0.000,B 0.000,C 180.000,E1 0.000} C_DIS
LIN {X -21.170,Y 45.230,Z 290.000,A 0.000,B 0.000,C 180.000,E1 0.000} C_DIS
LIN {X -23.465,Y 44.082,Z 290.000,A 0.000,B 0.000,C 180.000,E1 0.000} C_DIS
LIN {X -25.709,Y 42.812,Z 290.000,A 0.000,B 0.000,C 180.000,E1 0.000} C_DIS
LIN {X -27.882,Y 41.431,Z 290.000,A 0.000,B 0.000,C 180.000,E1 0.000} C_DIS
LIN {X -29.974,Y 39.943,Z 290.000,A 0.000,B 0.000,C 180.000,E1 0.000} C_DIS
LIN {X -31.988,Y 38.349,Z 290.000,A 0.000,B 0.000,C 180.000,E1 0.000} C_DIS
LIN {X -33.920,Y 36.650,Z 290.000,A 0.000,B 0.000,C 180.000,E1 0.000} C_DIS
LIN {X -35.767,Y 34.851,Z 290.000,A 0.000,B 0.000,C 180.000,E1 0.000} C_DIS
LIN {X -37.509,Y 32.969,Z 290.000,A 0.000,B 0.000,C 180.000,E1 0.000} C_DIS
LIN {X -39.156,Y 30.993,Z 290.000,A 0.000,B 0.000,C 180.000,E1 0.000} C_DIS
LIN {X -40.701,Y 28.935,Z 290.000,A 0.000,B 0.000,C 180.000,E1 0.000} C_DIS
LIN {X -42.137,Y 26.801,Z 290.000,A 0.000,B 0.000,C 180.000,E1 0.000} C_DIS
LIN {X -43.463,Y 24.594,Z 290.000,A 0.000,B 0.000,C 180.000,E1 0.000} C_DIS
LIN {X -44.669,Y 22.330,Z 290.000,A 0.000,B 0.000,C 180.000,E1 0.000} C_DIS
LIN {X -45.758,Y 20.000,Z 290.000,A 0.000,B 0.000,C 180.000,E1 0.000} C_DIS
LIN {X -46.729,Y 17.614,Z 290.000,A 0.000,B 0.000,C 180.000,E1 0.000} C_DIS
LIN {X -47.573,Y 15.187,Z 290.000,A 0.000,B 0.000,C 180.000,E1 0.000} C_DIS
LIN {X -48.292,Y 12.718,Z 290.000,A 0.000,B 0.000,C 180.000,E1 0.000} C_DIS
LIN {X -48.883,Y 10.214,Z 290.000,A 0.000,B 0.000,C 180.000,E1 0.000} C_DIS
LIN {X -49.344,Y 7.684,Z 290.000,A 0.000,B 0.000,C 180.000,E1 0.000} C_DIS
LIN {X -49.673,Y 5.144,Z 290.000,A 0.000,B 0.000,C 180.000,E1 0.000} C_DIS
LIN {X -49.873,Y 2.567,Z 290.000,A 0.000,B 0.000,C 180.000,E1 0.000} C_DIS
LIN {X -49.939,Y 0.000,Z 290.000,A 0.000,B 0.000,C 180.000,E1 0.000} C_DIS
LIN {X -49.873,Y -2.567,Z 290.000,A 0.000,B 0.000,C 180.000,E1 0.000} C_DIS
LIN {X -49.674,Y -5.134,Z 290.000,A 0.000,B 0.000,C 180.000,E1 0.000} C_DIS
;rapid-leaky
$VEL.CP=0.3
LIN {X -32.154,Y 0.728,Z 290.000,A 0.000,B 0.000,C 180.000,E1 0.000} C_DIS
;bead-solid_infill
$VEL.CP=0.16
LIN {X 0.736,Y -32.162,Z 290.000,A 0.000,B 0.000,C 180.000,E1 0.000} C_DIS
LIN {X 0.828,Y -32.162,Z 290.000,A 0.000,B 0.000,C 180.000,E1 0.000} C_DIS
LIN {X 2.480,Y -32.077,Z 290.000,A 0.000,B 0.000,C 180.000,E1 0.000} C_DIS
LIN {X 4.129,Y -31.906,Z 290.000,A 0.000,B 0.000,C 180.000,E1 0.000} C_DIS
LIN {X 5.773,Y -31.650,Z 290.000,A 0.000,B 0.000,C 180.000,E1 0.000} C_DIS
LIN {X 7.391,Y -31.312,Z 290.000,A 0.000,B 0.000,C 180.000,E1 0.000} C_DIS
LIN {X 8.989,Y -30.891,Z 290.000,A 0.000,B 0.000,C 180.000,E1 0.000} C_DIS
LIN {X 10.572,Y -30.386,Z 290.000,A 0.000,B 0.000,C 180.000,E1 0.000} C_DIS
LIN {X 12.124,Y -29.801,Z 290.000,A 0.000,B 0.000,C 180.000,E1 0.000} C_DIS
LIN {X 13.638,Y -29.140,Z 290.000,A 0.000,B 0.000,C 180.000,E1 0.000} C_DIS
LIN {X 15.113,Y -28.402,Z 290.000,A 0.000,B 0.000,C 180.000,E1 0.000} C_DIS
LIN {X 16.565,Y -27.580,Z 290.000,A 0.000,B 0.000,C 180.000,E1 0.000} C_DIS
LIN {X 17.966,Y -26.689,Z 290.000,A 0.000,B 0.000,C 180.000,E1 0.000} C_DIS
LIN {X 19.310,Y -25.734,Z 290.000,A 0.000,B 0.000,C 180.000,E1 0.000} C_DIS
LIN {X 20.605,Y -24.709,Z 290.000,A 0.000,B 0.000,C 180.000,E1 0.000} C_DIS
LIN {X 21.852,Y -23.612,Z 290.000,A 0.000,B 0.000,C 180.000,E1 0.000} C_DIS
LIN {X 22.728,Y -22.759,Z 290.000,A 0.000,B 0.000,C 180.000,E1 0.000} C_DIS
LIN {X -22.759,Y 22.729,Z 290.000,A 0.000,B 0.000,C 180.000,E1 0.000} C_DIS
LIN {X -21.852,Y 23.612,Z 290.000,A 0.000,B 0.000,C 180.000,E1 0.000} C_DIS
LIN {X -20.605,Y 24.709,Z 290.000,A 0.000,B 0.000,C 180.000,E1 0.000} C_DIS
LIN {X -19.310,Y 25.734,Z 290.000,A 0.000,B 0.000,C 180.000,E1 0.000} C_DIS
LIN {X -17.966,Y 26.689,Z 290.000,A 0.000,B 0.000,C 180.000,E1 0.000} C_DIS
LIN {X -16.565,Y 27.580,Z 290.000,A 0.000,B 0.000,C 180.000,E1 0.000} C_DIS
LIN {X -15.113,Y 28.402,Z 290.000,A 0.000,B 0.000,C 180.000,E1 0.000} C_DIS
LIN {X -13.638,Y 29.140,Z 290.000,A 0.000,B 0.000,C 180.000,E1 0.000} C_DIS
LIN {X -12.124,Y 29.801,Z 290.000,A 0.000,B 0.000,C 180.000,E1 0.000} C_DIS
LIN {X -10.572,Y 30.386,Z 290.000,A 0.000,B 0.000,C 180.000,E1 0.000} C_DIS
LIN {X -8.989,Y 30.891,Z 290.000,A 0.000,B 0.000,C 180.000,E1 0.000} C_DIS
LIN {X -7.391,Y 31.312,Z 290.000,A 0.000,B 0.000,C 180.000,E1 0.000} C_DIS
LIN {X -5.773,Y 31.650,Z 290.000,A 0.000,B 0.000,C 180.000,E1 0.000} C_DIS
LIN {X -4.129,Y 31.906,Z 290.000,A 0.000,B 0.000,C 180.000,E1 0.000} C_DIS
LIN {X -2.480,Y 32.077,Z 290.000,A 0.000,B 0.000,C 180.000,E1 0.000} C_DIS
LIN {X -0.828,Y 32.162,Z 290.000,A 0.000,B 0.000,C 180.000,E1 0.000} C_DIS
LIN {X -0.797,Y 32.162,Z 290.000,A 0.000,B 0.000,C 180.000,E1 0.000} C_DIS
LIN {X 32.153,Y -0.788,Z 290.000,A 0.000,B 0.000,C 180.000,E1 0.000} C_DIS
$VEL.CP=0.3
LIN {X 32.153,Y -0.788,Z 290.000,A 0.000,B 0.000,C 180.000,E1 0.000} C_DIS
;part 1 complete
;move to park position
LIN {X 32.153,Y -0.788,Z 400.000,A 0.000,B 0.000,C 180.000,E1 0.000} C_DIS
LIN {X 200.000,Y 200.000,Z 400.000,A 0.000,B 0.000,C 180.000,E1 0.000} C_DIS
EXTRUDER_STATE=FALSE
home_cycle()
;PTP XHOME
;--------------------------------
;--------------------------------
;ENDFOLD
END
